LIN {X 0,Y 466.62,Z 631.984,A -85,B 0,C 180,E1 -7650.863,E2 -7650.863} C_VEL
LIN {X 0,Y 466.694,Z 631.335,A -85,B 0,C 180,E1 -7651.726,E2 -7651.726} C_VEL
LIN {X 0,Y 466.71,Z 630.282,A -85,B 0,C 180,E1 -7652.589,E2 -7652.589} C_VEL
LIN {X 0,Y 466.73,Z 628.811,A -85,B 0,C 180,E1 -7653.453,E2 -7653.453} C_VEL
LIN {X 0,Y 466.701,Z 625.736,A -85,B 0,C 180,E1 -7654.751,E2 -7654.751} C_VEL
LIN {X 0,Y 466.773,Z 621.588,A -85,B 0,C 180,E1 -7656.05,E2 -7656.05} C_VEL
LIN {X 0,Y 466.928,Z 615.211,A -85,B 0,C 180,E1 -7657.568,E2 -7657.568} C_VEL
LIN {X 0,Y 467.142,Z 608.264,A -85,B 0,C 180,E1 -7658.871,E2 -7658.871} C_VEL
LIN {X 0,Y 467.463,Z 599.648,A -85,B 0,C 180,E1 -7660.175,E2 -7660.175} C_VEL
LIN {X 0,Y 467.909,Z 590.815,A -85,B 0,C 180,E1 -7661.26,E2 -7661.26} C_VEL
LIN {X 0,Y 468.338,Z 580.643,A -85,B 0,C 180,E1 -7662.287,E2 -7662.287} C_VEL
LIN {X 0,Y 468.829,Z 569.32,A -85,B 0,C 180,E1 -7663.215,E2 -7663.215} C_VEL
LIN {X 0,Y 469.286,Z 557.554,A -85,B 0,C 180,E1 -7663.975,E2 -7663.975} C_VEL
LIN {X 0,Y 469.739,Z 544.43,A -85,B 0,C 180,E1 -7664.624,E2 -7664.624} C_VEL
LIN {X 0,Y 468.125,Z 531.649,A -85,B 0,C 180,E1 -7665.143,E2 -7665.143} C_VEL
LIN {X 0,Y 467.02,Z 523.223,A -85,B 0,C 180,E1 -7665.409,E2 -7665.409} C_VEL
LIN {X 0,Y 467.168,Z 513.678,A -85,B 0,C 180,E1 -7668.601,E2 -7668.601} C_VEL
LIN {X 0,Y 467.391,Z 504.9,A -85,B 0,C 180,E1 -7671.617,E2 -7671.617} C_VEL
LIN {X 0,Y 467.664,Z 495.775,A -85,B 0,C 180,E1 -7674.884,E2 -7674.884} C_VEL
LIN {X 0,Y 468.021,Z 488.237,A -85,B 0,C 180,E1 -7677.743,E2 -7677.743} C_VEL
LIN {X 0,Y 468.559,Z 479.713,A -85,B 0,C 180,E1 -7681.245,E2 -7681.245} C_VEL
LIN {X 0,Y 469.039,Z 474.432,A -85,B 0,C 180,E1 -7683.67,E2 -7683.67} C_VEL
LIN {X 0,Y 469.375,Z 469.859,A -85,B 0,C 180,E1 -7686.046,E2 -7686.046} C_VEL
LIN {X 0,Y 469.096,Z 466.887,A -85,B 0,C 180,E1 -7687.899,E2 -7687.899} C_VEL
LIN {X 0,Y 468.575,Z 463.943,A -85,B 0,C 180,E1 -7690.162,E2 -7690.162} C_VEL
LIN {X 0,Y 468.164,Z 461.563,A -85,B 0,C 180,E1 -7692.644,E2 -7692.644} C_VEL
LIN {X 0,Y 467.906,Z 460.071,A -85,B 0,C 180,E1 -7695.094,E2 -7695.094} C_VEL
LIN {X 0,Y 467.787,Z 459.398,A -85,B 0,C 180,E1 -7697.462,E2 -7697.462} C_VEL
LIN {X 0,Y 467.762,Z 459.412,A -85,B 0,C 180,E1 -7700.02,E2 -7700.02} C_VEL
LIN {X 0,Y 467.837,Z 460.213,A -85,B 0,C 180,E1 -7703.066,E2 -7703.066} C_VEL
LIN {X 0,Y 467.816,Z 461.445,A -85,B 0,C 180,E1 -7705.717,E2 -7705.717} C_VEL
LIN {X 0,Y 467.647,Z 462.959,A -85,B 0,C 180,E1 -7708.265,E2 -7708.265} C_VEL
LIN {X 0,Y 467.464,Z 465.049,A -85,B 0,C 180,E1 -7711.243,E2 -7711.243} C_VEL
LIN {X 0,Y 467.288,Z 467.552,A -85,B 0,C 180,E1 -7714.476,E2 -7714.476} C_VEL
LIN {X 0,Y 467.169,Z 469.646,A -85,B 0,C 180,E1 -7716.975,E2 -7716.975} C_VEL
LIN {X 0,Y 467.058,Z 472.089,A -85,B 0,C 180,E1 -7719.752,E2 -7719.752} C_VEL
LIN {X 0,Y 466.99,Z 474.598,A -85,B 0,C 180,E1 -7722.483,E2 -7722.483} C_VEL
LIN {X 0,Y 467.017,Z 476.743,A -85,B 0,C 180,E1 -7724.739,E2 -7724.739} C_VEL
LIN {X 0,Y 469.978,Z 489.42,A -85,B 0,C 180,E1 -7725.273,E2 -7725.273} C_VEL
LIN {X 0,Y 470.134,Z 495.785,A -85,B 0,C 180,E1 -7725.555,E2 -7725.555} C_VEL
LIN {X 0,Y 469.76,Z 507.117,A -85,B 0,C 180,E1 -7726.151,E2 -7726.151} C_VEL
LIN {X 0,Y 469.317,Z 518.894,A -85,B 0,C 180,E1 -7726.955,E2 -7726.955} C_VEL
LIN {X 0,Y 468.819,Z 529.714,A -85,B 0,C 180,E1 -7727.885,E2 -7727.885} C_VEL
LIN {X 0,Y 468.295,Z 539.912,A -85,B 0,C 180,E1 -7728.969,E2 -7728.969} C_VEL
LIN {X 0,Y 467.847,Z 549.675,A -85,B 0,C 180,E1 -7730.271,E2 -7730.271} C_VEL
LIN {X 0,Y 467.45,Z 557.526,A -85,B 0,C 180,E1 -7731.571,E2 -7731.571} C_VEL
LIN {X 0,Y 467.22,Z 562.822,A -85,B 0,C 180,E1 -7732.654,E2 -7732.654} C_VEL
LIN {X 0,Y 467.057,Z 567.987,A -85,B 0,C 180,E1 -7733.954,E2 -7733.954} C_VEL
LIN {X 0,Y 466.887,Z 571.984,A -85,B 0,C 180,E1 -7735.251,E2 -7735.251} C_VEL
LIN {X 0,Y 466.794,Z 574.921,A -85,B 0,C 180,E1 -7736.548,E2 -7736.548} C_VEL
LIN {X 0,Y 466.81,Z 576.332,A -85,B 0,C 180,E1 -7737.411,E2 -7737.411} C_VEL
LIN {X 0,Y 466.62,Z 577.923,A -85,B 0,C 180,E1 -7739.137,E2 -7739.137} C_VEL
LIN {X 0,Y 466.6,Z 578.133,A -85,B 0,C 180,E1 -7740,E2 -7740} C_VEL
LIN {X 0,Y 466.62,Z 577.913,A -85,B 0,C 180,E1 -7740.863,E2 -7740.863} C_VEL
LIN {X 0,Y 466.79,Z 576.267,A -85,B 0,C 180,E1 -7742.589,E2 -7742.589} C_VEL
LIN {X 0,Y 466.786,Z 574.855,A -85,B 0,C 180,E1 -7743.453,E2 -7743.453} C_VEL
LIN {X 0,Y 466.861,Z 571.894,A -85,B 0,C 180,E1 -7744.75,E2 -7744.75} C_VEL
LIN {X 0,Y 467.046,Z 567.886,A -85,B 0,C 180,E1 -7746.047,E2 -7746.047} C_VEL
LIN {X 0,Y 467.174,Z 562.727,A -85,B 0,C 180,E1 -7747.347,E2 -7747.347} C_VEL
LIN {X 0,Y 467.431,Z 556.22,A -85,B 0,C 180,E1 -7748.648,E2 -7748.648} C_VEL
LIN {X 0,Y 467.789,Z 548.123,A -85,B 0,C 180,E1 -7749.949,E2 -7749.949} C_VEL
LIN {X 0,Y 468.17,Z 539.866,A -85,B 0,C 180,E1 -7751.035,E2 -7751.035} C_VEL
LIN {X 0,Y 468.738,Z 529.781,A -85,B 0,C 180,E1 -7752.117,E2 -7752.117} C_VEL
LIN {X 0,Y 469.143,Z 518.266,A -85,B 0,C 180,E1 -7753.107,E2 -7753.107} C_VEL
LIN {X 0,Y 469.555,Z 507.32,A -85,B 0,C 180,E1 -7753.856,E2 -7753.856} C_VEL
LIN {X 0,Y 469.986,Z 495.028,A -85,B 0,C 180,E1 -7754.506,E2 -7754.506} C_VEL
LIN {X 0,Y 469.852,Z 489.361,A -85,B 0,C 180,E1 -7754.754,E2 -7754.754} C_VEL
LIN {X 0,Y 467.68,Z 478.772,A -85,B 0,C 180,E1 -7755.187,E2 -7755.187} C_VEL
LIN {X 0,Y 466.852,Z 474.833,A -85,B 0,C 180,E1 -7755.323,E2 -7755.323} C_VEL
LIN {X 0,Y 466.83,Z 471.352,A -85,B 0,C 180,E1 -7758.476,E2 -7758.476} C_VEL
LIN {X 0,Y 466.807,Z 468.406,A -85,B 0,C 180,E1 -7761.182,E2 -7761.182} C_VEL
LIN {X 0,Y 466.863,Z 465.394,A -85,B 0,C 180,E1 -7763.982,E2 -7763.982} C_VEL
LIN {X 0,Y 466.949,Z 462.367,A -85,B 0,C 180,E1 -7766.842,E2 -7766.842} C_VEL
LIN {X 0,Y 466.958,Z 459.297,A -85,B 0,C 180,E1 -7769.78,E2 -7769.78} C_VEL
LIN {X 0,Y 467.012,Z 458.315,A -85,B 0,C 180,E1 -7770.931,E2 -7770.931} C_VEL
LIN {X 0,Y 467.392,Z 458.268,A -85,B 0,C 180,E1 -7774.206,E2 -7774.206} C_VEL
LIN {X 0,Y 467.544,Z 458.245,A -85,B 0,C 180,E1 -7777.185,E2 -7777.185} C_VEL
LIN {X 0,Y 467.582,Z 458.242,A -85,B 0,C 180,E1 -7780.265,E2 -7780.265} C_VEL
LIN {X 0,Y 467.591,Z 458.241,A -85,B 0,C 180,E1 -7782.567,E2 -7782.567} C_VEL
LIN {X 0,Y 467.571,Z 458.241,A -85,B 0,C 180,E1 -7785.053,E2 -7785.053} C_VEL
LIN {X 0,Y 467.594,Z 458.239,A -85,B 0,C 180,E1 -7787.44,E2 -7787.44} C_VEL
LIN {X 0,Y 467.587,Z 458.241,A -85,B 0,C 180,E1 -7790.855,E2 -7790.855} C_VEL
LIN {X 0,Y 467.565,Z 458.245,A -85,B 0,C 180,E1 -7794.261,E2 -7794.261} C_VEL
LIN {X 0,Y 467.587,Z 458.241,A -85,B 0,C 180,E1 -7797.321,E2 -7797.321} C_VEL
LIN {X 0,Y 467.573,Z 458.241,A -85,B 0,C 180,E1 -7800.668,E2 -7800.668} C_VEL
LIN {X 0,Y 467.622,Z 458.237,A -85,B 0,C 180,E1 -7803.2,E2 -7803.2} C_VEL
LIN {X 0,Y 467.598,Z 458.241,A -85,B 0,C 180,E1 -7806.468,E2 -7806.468} C_VEL
LIN {X 0,Y 467.629,Z 458.238,A -85,B 0,C 180,E1 -7809.777,E2 -7809.777} C_VEL
LIN {X 0,Y 467.628,Z 458.236,A -85,B 0,C 180,E1 -7811.423,E2 -7811.423} C_VEL
LIN {X 0,Y 466.988,Z 458.317,A -85,B 0,C 180,E1 -7812.142,E2 -7812.142} C_VEL
LIN {X 0,Y 464.137,Z 458.669,A -85,B 0,C 180,E1 -7813.31,E2 -7813.31} C_VEL
LIN {X 0,Y 461.703,Z 458.976,A -85,B 0,C 180,E1 -7814.251,E2 -7814.251} C_VEL
LIN {X 0,Y 460.647,Z 459.103,A -85,B 0,C 180,E1 -7814.979,E2 -7814.979} C_VEL
LIN {X 0,Y 460.557,Z 459.114,A -85,B 0,C 180,E1 -7815.226,E2 -7815.226} C_VEL
LIN {X 0,Y 460.616,Z 459.111,A -85,B 0,C 180,E1 -7818.559,E2 -7818.559} C_VEL
LIN {X 0,Y 460.671,Z 459.105,A -85,B 0,C 180,E1 -7822.108,E2 -7822.108} C_VEL
LIN {X 0,Y 460.702,Z 459.099,A -85,B 0,C 180,E1 -7824.748,E2 -7824.748} C_VEL
LIN {X 0,Y 460.805,Z 459.085,A -85,B 0,C 180,E1 -7827.377,E2 -7827.377} C_VEL
LIN {X 0,Y 460.859,Z 459.081,A -85,B 0,C 180,E1 -7830,E2 -7830} C_VEL
LIN {X 0,Y 460.805,Z 459.087,A -85,B 0,C 180,E1 -7832.622,E2 -7832.622} C_VEL
LIN {X 0,Y 460.69,Z 459.102,A -85,B 0,C 180,E1 -7836.13,E2 -7836.13} C_VEL
LIN {X 0,Y 460.634,Z 459.107,A -85,B 0,C 180,E1 -7838.776,E2 -7838.776} C_VEL
LIN {X 0,Y 460.619,Z 459.109,A -85,B 0,C 180,E1 -7842.445,E2 -7842.445} C_VEL
LIN {X 0,Y 460.605,Z 459.111,A -85,B 0,C 180,E1 -7845.997,E2 -7845.997} C_VEL
LIN {X 0,Y 460.576,Z 459.114,A -85,B 0,C 180,E1 -7848.901,E2 -7848.901} C_VEL
LIN {X 0,Y 460.521,Z 459.121,A -85,B 0,C 180,E1 -7851.485,E2 -7851.485} C_VEL
LIN {X 0,Y 460.546,Z 459.119,A -85,B 0,C 180,E1 -7854.332,E2 -7854.332} C_VEL
LIN {X 0,Y 460.577,Z 459.112,A -85,B 0,C 180,E1 -7857.243,E2 -7857.243} C_VEL
LIN {X 0,Y 460.515,Z 459.121,A -85,B 0,C 180,E1 -7860.24,E2 -7860.24} C_VEL
LIN {X 0,Y 460.533,Z 459.119,A -85,B 0,C 180,E1 -7863.324,E2 -7863.324} C_VEL
LIN {X 0,Y 460.482,Z 459.124,A -85,B 0,C 180,E1 -7866.529,E2 -7866.529} C_VEL
LIN {X 0,Y 460.548,Z 459.118,A -85,B 0,C 180,E1 -7868.897,E2 -7868.897} C_VEL
LIN {X 0,Y 460.526,Z 459.12,A -85,B 0,C 180,E1 -7872.181,E2 -7872.181} C_VEL
LIN {X 0,Y 460.523,Z 459.122,A -85,B 0,C 180,E1 -7875.412,E2 -7875.412} C_VEL
LIN {X 0,Y 460.538,Z 459.118,A -85,B 0,C 180,E1 -7878.397,E2 -7878.397} C_VEL
LIN {X 0,Y 460.521,Z 459.122,A -85,B 0,C 180,E1 -7881.266,E2 -7881.266} C_VEL
LIN {X 0,Y 460.516,Z 459.121,A -85,B 0,C 180,E1 -7884.554,E2 -7884.554} C_VEL
LIN {X 0,Y 460.534,Z 459.121,A -85,B 0,C 180,E1 -7887.715,E2 -7887.715} C_VEL
LIN {X 0,Y 460.542,Z 459.119,A -85,B 0,C 180,E1 -7890.769,E2 -7890.769} C_VEL
LIN {X 0,Y 460.565,Z 459.118,A -85,B 0,C 180,E1 -7893.734,E2 -7893.734} C_VEL
LIN {X 0,Y 460.547,Z 459.118,A -85,B 0,C 180,E1 -7896.624,E2 -7896.624} C_VEL
LIN {X 0,Y 460.554,Z 459.117,A -85,B 0,C 180,E1 -7899.453,E2 -7899.453} C_VEL
LIN {X 0,Y 460.561,Z 459.114,A -85,B 0,C 180,E1 -7902.23,E2 -7902.23} C_VEL
LIN {X 0,Y 460.567,Z 459.117,A -85,B 0,C 180,E1 -7904.965,E2 -7904.965} C_VEL
LIN {X 0,Y 460.613,Z 459.106,A -85,B 0,C 180,E1 -7908.559,E2 -7908.559} C_VEL
LIN {X 0,Y 460.696,Z 459.101,A -85,B 0,C 180,E1 -7912.108,E2 -7912.108} C_VEL
LIN {X 0,Y 460.698,Z 459.097,A -85,B 0,C 180,E1 -7914.748,E2 -7914.748} C_VEL
LIN {X 0,Y 460.825,Z 459.085,A -85,B 0,C 180,E1 -7917.377,E2 -7917.377} C_VEL
LIN {X 0,Y 460.855,Z 459.081,A -85,B 0,C 180,E1 -7920,E2 -7920} C_VEL
LIN {X 0,Y 460.801,Z 459.084,A -85,B 0,C 180,E1 -7922.622,E2 -7922.622} C_VEL
LIN {X 0,Y 460.711,Z 459.098,A -85,B 0,C 180,E1 -7926.13,E2 -7926.13} C_VEL
LIN {X 0,Y 460.629,Z 459.106,A -85,B 0,C 180,E1 -7928.776,E2 -7928.776} C_VEL
LIN {X 0,Y 460.614,Z 459.109,A -85,B 0,C 180,E1 -7932.445,E2 -7932.445} C_VEL
LIN {X 0,Y 460.601,Z 459.111,A -85,B 0,C 180,E1 -7935.997,E2 -7935.997} C_VEL
LIN {X 0,Y 460.572,Z 459.115,A -85,B 0,C 180,E1 -7938.902,E2 -7938.902} C_VEL
LIN {X 0,Y 460.516,Z 459.122,A -85,B 0,C 180,E1 -7941.486,E2 -7941.486} C_VEL
LIN {X 0,Y 460.543,Z 459.115,A -85,B 0,C 180,E1 -7944.332,E2 -7944.332} C_VEL
LIN {X 0,Y 460.58,Z 459.114,A -85,B 0,C 180,E1 -7947.243,E2 -7947.243} C_VEL
LIN {X 0,Y 460.511,Z 459.121,A -85,B 0,C 180,E1 -7950.24,E2 -7950.24} C_VEL
LIN {X 0,Y 460.529,Z 459.121,A -85,B 0,C 180,E1 -7953.325,E2 -7953.325} C_VEL
LIN {X 0,Y 460.479,Z 459.127,A -85,B 0,C 180,E1 -7956.529,E2 -7956.529} C_VEL
LIN {X 0,Y 460.545,Z 459.117,A -85,B 0,C 180,E1 -7958.898,E2 -7958.898} C_VEL
LIN {X 0,Y 460.547,Z 459.118,A -85,B 0,C 180,E1 -7962.179,E2 -7962.179} C_VEL
LIN {X 0,Y 460.514,Z 459.128,A -85,B 0,C 180,E1 -7965.411,E2 -7965.411} C_VEL
LIN {X 0,Y 460.532,Z 459.124,A -85,B 0,C 180,E1 -7968.398,E2 -7968.398} C_VEL
LIN {X 0,Y 460.565,Z 459.206,A -85,B 0,C 180,E1 -7969.188,E2 -7969.188} C_VEL
LIN {X 0,Y 461.793,Z 466.092,A -85,B 0,C 180,E1 -7972.315,E2 -7972.315} C_VEL
LIN {X 0,Y 462.377,Z 470.478,A -85,B 0,C 180,E1 -7974.209,E2 -7974.209} C_VEL
LIN {X 0,Y 462.014,Z 476.847,A -85,B 0,C 180,E1 -7976.796,E2 -7976.796} C_VEL
LIN {X 0,Y 461.551,Z 484.581,A -85,B 0,C 180,E1 -7979.835,E2 -7979.835} C_VEL
LIN {X 0,Y 461.107,Z 492.34,A -85,B 0,C 180,E1 -7982.791,E2 -7982.791} C_VEL
LIN {X 0,Y 460.773,Z 500.11,A -85,B 0,C 180,E1 -7985.681,E2 -7985.681} C_VEL
LIN {X 0,Y 460.386,Z 509.336,A -85,B 0,C 180,E1 -7989.025,E2 -7989.025} C_VEL
LIN {X 0,Y 460.159,Z 517.005,A -85,B 0,C 180,E1 -7991.754,E2 -7991.754} C_VEL
LIN {X 0,Y 460.033,Z 524.604,A -85,B 0,C 180,E1 -7994.406,E2 -7994.406} C_VEL
LIN {X 0,Y 461.907,Z 538.263,A -85,B 0,C 180,E1 -7994.853,E2 -7994.853} C_VEL
LIN {X 0,Y 462.917,Z 546.399,A -85,B 0,C 180,E1 -7995.212,E2 -7995.212} C_VEL
LIN {X 0,Y 462.482,Z 558.305,A -85,B 0,C 180,E1 -7995.816,E2 -7995.816} C_VEL
LIN {X 0,Y 461.956,Z 569.987,A -85,B 0,C 180,E1 -7996.585,E2 -7996.585} C_VEL
LIN {X 0,Y 461.407,Z 581.292,A -85,B 0,C 180,E1 -7997.534,E2 -7997.534} C_VEL
LIN {X 0,Y 460.931,Z 591.248,A -85,B 0,C 180,E1 -7998.567,E2 -7998.567} C_VEL
LIN {X 0,Y 460.462,Z 599.965,A -85,B 0,C 180,E1 -7999.669,E2 -7999.669} C_VEL
LIN {X 0,Y 460.108,Z 608.449,A -85,B 0,C 180,E1 -8000.993,E2 -8000.993} C_VEL
LIN {X 0,Y 459.867,Z 615.276,A -85,B 0,C 180,E1 -8002.315,E2 -8002.315} C_VEL
LIN {X 0,Y 459.677,Z 621.541,A -85,B 0,C 180,E1 -8003.856,E2 -8003.856} C_VEL
LIN {X 0,Y 459.631,Z 625.603,A -85,B 0,C 180,E1 -8005.176,E2 -8005.176} C_VEL
LIN {X 0,Y 459.627,Z 628.592,A -85,B 0,C 180,E1 -8006.494,E2 -8006.494} C_VEL
LIN {X 0,Y 459.621,Z 630.019,A -85,B 0,C 180,E1 -8007.371,E2 -8007.371} C_VEL
LIN {X 0,Y 459.629,Z 631.023,A -85,B 0,C 180,E1 -8008.248,E2 -8008.248} C_VEL
LIN {X 0,Y 459.553,Z 631.62,A -85,B 0,C 180,E1 -8009.124,E2 -8009.124} C_VEL
LIN {X 0,Y 459.529,Z 631.819,A -85,B 0,C 180,E1 -8010,E2 -8010} C_VEL
LIN {X 0,Y 459.553,Z 631.571,A -85,B 0,C 180,E1 -8010.876,E2 -8010.876} C_VEL
LIN {X 0,Y 459.631,Z 630.919,A -85,B 0,C 180,E1 -8011.753,E2 -8011.753} C_VEL
LIN {X 0,Y 459.63,Z 629.858,A -85,B 0,C 180,E1 -8012.629,E2 -8012.629} C_VEL
LIN {X 0,Y 459.643,Z 628.379,A -85,B 0,C 180,E1 -8013.507,E2 -8013.507} C_VEL
LIN {X 0,Y 459.632,Z 625.289,A -85,B 0,C 180,E1 -8014.824,E2 -8014.824} C_VEL
LIN {X 0,Y 459.714,Z 620.037,A -85,B 0,C 180,E1 -8016.431,E2 -8016.431} C_VEL
LIN {X 0,Y 459.895,Z 613.684,A -85,B 0,C 180,E1 -8017.905,E2 -8017.905} C_VEL
LIN {X 0,Y 460.181,Z 606.485,A -85,B 0,C 180,E1 -8019.228,E2 -8019.228} C_VEL
LIN {X 0,Y 460.507,Z 597.482,A -85,B 0,C 180,E1 -8020.553,E2 -8020.553} C_VEL
LIN {X 0,Y 461.071,Z 587.326,A -85,B 0,C 180,E1 -8021.764,E2 -8021.764} C_VEL
LIN {X 0,Y 461.488,Z 576.916,A -85,B 0,C 180,E1 -8022.767,E2 -8022.767} C_VEL
LIN {X 0,Y 462.034,Z 565.747,A -85,B 0,C 180,E1 -8023.637,E2 -8023.637} C_VEL
LIN {X 0,Y 462.589,Z 553.269,A -85,B 0,C 180,E1 -8024.406,E2 -8024.406} C_VEL
LIN {X 0,Y 462.819,Z 545.368,A -85,B 0,C 180,E1 -8024.792,E2 -8024.792} C_VEL
LIN {X 0,Y 461.169,Z 531.714,A -85,B 0,C 180,E1 -8025.377,E2 -8025.377} C_VEL
LIN {X 0,Y 459.944,Z 522.74,A -85,B 0,C 180,E1 -8025.664,E2 -8025.664} C_VEL
LIN {X 0,Y 460.125,Z 512.626,A -85,B 0,C 180,E1 -8029.125,E2 -8029.125} C_VEL
LIN {X 0,Y 460.346,Z 504.578,A -85,B 0,C 180,E1 -8031.965,E2 -8031.965} C_VEL
LIN {X 0,Y 460.679,Z 495.558,A -85,B 0,C 180,E1 -8035.288,E2 -8035.288} C_VEL
LIN {X 0,Y 461.042,Z 488.122,A -85,B 0,C 180,E1 -8038.201,E2 -8038.201} C_VEL
LIN {X 0,Y 461.592,Z 480.372,A -85,B 0,C 180,E1 -8041.501,E2 -8041.501} C_VEL
LIN {X 0,Y 462.144,Z 474.635,A -85,B 0,C 180,E1 -8044.241,E2 -8044.241} C_VEL
LIN {X 0,Y 462.399,Z 470.78,A -85,B 0,C 180,E1 -8046.353,E2 -8046.353} C_VEL
LIN {X 0,Y 462.013,Z 467.441,A -85,B 0,C 180,E1 -8048.586,E2 -8048.586} C_VEL
LIN {X 0,Y 461.529,Z 464.7,A -85,B 0,C 180,E1 -8050.904,E2 -8050.904} C_VEL
LIN {X 0,Y 461.142,Z 462.652,A -85,B 0,C 180,E1 -8053.3,E2 -8053.3} C_VEL
LIN {X 0,Y 460.922,Z 461.348,A -85,B 0,C 180,E1 -8055.778,E2 -8055.778} C_VEL
LIN {X 0,Y 460.826,Z 460.803,A -85,B 0,C 180,E1 -8058.357,E2 -8058.357} C_VEL
LIN {X 0,Y 460.804,Z 461.042,A -85,B 0,C 180,E1 -8061.295,E2 -8061.295} C_VEL
LIN {X 0,Y 460.87,Z 461.851,A -85,B 0,C 180,E1 -8063.923,E2 -8063.923} C_VEL
LIN {X 0,Y 460.746,Z 463.376,A -85,B 0,C 180,E1 -8067.029,E2 -8067.029} C_VEL
LIN {X 0,Y 460.511,Z 465.551,A -85,B 0,C 180,E1 -8070.447,E2 -8070.447} C_VEL
LIN {X 0,Y 460.288,Z 467.945,A -85,B 0,C 180,E1 -8073.718,E2 -8073.718} C_VEL
LIN {X 0,Y 460.182,Z 470.267,A -85,B 0,C 180,E1 -8076.604,E2 -8076.604} C_VEL
LIN {X 0,Y 460.019,Z 472.686,A -85,B 0,C 180,E1 -8079.428,E2 -8079.428} C_VEL
LIN {X 0,Y 459.946,Z 475.184,A -85,B 0,C 180,E1 -8082.206,E2 -8082.206} C_VEL
LIN {X 0,Y 459.946,Z 477.301,A -85,B 0,C 180,E1 -8084.471,E2 -8084.471} C_VEL
LIN {X 0,Y 463.097,Z 490.22,A -85,B 0,C 180,E1 -8085.049,E2 -8085.049} C_VEL
LIN {X 0,Y 463.31,Z 495.315,A -85,B 0,C 180,E1 -8085.281,E2 -8085.281} C_VEL
LIN {X 0,Y 462.917,Z 507.758,A -85,B 0,C 180,E1 -8085.942,E2 -8085.942} C_VEL
LIN {X 0,Y 462.437,Z 518.485,A -85,B 0,C 180,E1 -8086.677,E2 -8086.677} C_VEL
LIN {X 0,Y 461.906,Z 530.268,A -85,B 0,C 180,E1 -8087.701,E2 -8087.701} C_VEL
LIN {X 0,Y 461.344,Z 540.431,A -85,B 0,C 180,E1 -8088.8,E2 -8088.8} C_VEL
LIN {X 0,Y 460.868,Z 550.145,A -85,B 0,C 180,E1 -8090.122,E2 -8090.122} C_VEL
LIN {X 0,Y 460.438,Z 557.967,A -85,B 0,C 180,E1 -8091.442,E2 -8091.442} C_VEL
LIN {X 0,Y 460.186,Z 563.247,A -85,B 0,C 180,E1 -8092.541,E2 -8092.541} C_VEL
LIN {X 0,Y 460.016,Z 568.417,A -85,B 0,C 180,E1 -8093.861,E2 -8093.861} C_VEL
LIN {X 0,Y 459.83,Z 572.417,A -85,B 0,C 180,E1 -8095.178,E2 -8095.178} C_VEL
LIN {X 0,Y 459.733,Z 575.353,A -85,B 0,C 180,E1 -8096.494,E2 -8096.494} C_VEL
LIN {X 0,Y 459.736,Z 576.763,A -85,B 0,C 180,E1 -8097.372,E2 -8097.372} C_VEL
LIN {X 0,Y 459.554,Z 578.344,A -85,B 0,C 180,E1 -8099.124,E2 -8099.124} C_VEL
LIN {X 0,Y 459.531,Z 578.549,A -85,B 0,C 180,E1 -8100,E2 -8100} C_VEL
LIN {X 0,Y 459.554,Z 578.319,A -85,B 0,C 180,E1 -8100.876,E2 -8100.876} C_VEL
LIN {X 0,Y 459.637,Z 577.682,A -85,B 0,C 180,E1 -8101.753,E2 -8101.753} C_VEL
LIN {X 0,Y 459.705,Z 576.654,A -85,B 0,C 180,E1 -8102.629,E2 -8102.629} C_VEL
LIN {X 0,Y 459.726,Z 575.229,A -85,B 0,C 180,E1 -8103.506,E2 -8103.506} C_VEL
LIN {X 0,Y 459.79,Z 572.247,A -85,B 0,C 180,E1 -8104.823,E2 -8104.823} C_VEL
LIN {X 0,Y 460.005,Z 568.213,A -85,B 0,C 180,E1 -8106.14,E2 -8106.14} C_VEL
LIN {X 0,Y 460.157,Z 562.011,A -85,B 0,C 180,E1 -8107.68,E2 -8107.68} C_VEL
LIN {X 0,Y 460.504,Z 555.24,A -85,B 0,C 180,E1 -8109,E2 -8109} C_VEL
LIN {X 0,Y 460.886,Z 546.841,A -85,B 0,C 180,E1 -8110.322,E2 -8110.322} C_VEL
LIN {X 0,Y 461.275,Z 538.195,A -85,B 0,C 180,E1 -8111.424,E2 -8111.424} C_VEL
LIN {X 0,Y 461.901,Z 527.691,A -85,B 0,C 180,E1 -8112.512,E2 -8112.512} C_VEL
LIN {X 0,Y 462.279,Z 517.091,A -85,B 0,C 180,E1 -8113.406,E2 -8113.406} C_VEL
LIN {X 0,Y 462.749,Z 505.515,A -85,B 0,C 180,E1 -8114.176,E2 -8114.176} C_VEL
LIN {X 0,Y 463.204,Z 492.473,A -85,B 0,C 180,E1 -8114.835,E2 -8114.835} C_VEL
LIN {X 0,Y 461.989,Z 485.133,A -85,B 0,C 180,E1 -8115.169,E2 -8115.169} C_VEL
LIN {X 0,Y 459.762,Z 475.138,A -85,B 0,C 180,E1 -8115.574,E2 -8115.574} C_VEL
LIN {X 0,Y 459.736,Z 471.673,A -85,B 0,C 180,E1 -8118.725,E2 -8118.725} C_VEL
LIN {X 0,Y 459.744,Z 468.648,A -85,B 0,C 180,E1 -8121.524,E2 -8121.524} C_VEL
LIN {X 0,Y 459.805,Z 465.601,A -85,B 0,C 180,E1 -8124.374,E2 -8124.374} C_VEL
LIN {X 0,Y 459.917,Z 462.535,A -85,B 0,C 180,E1 -8127.286,E2 -8127.286} C_VEL
LIN {X 0,Y 459.904,Z 459.428,A -85,B 0,C 180,E1 -8130.285,E2 -8130.285} C_VEL
LIN {X 0,Y 460.173,Z 459.167,A -85,B 0,C 180,E1 -8132.861,E2 -8132.861} C_VEL
LIN {X 0,Y 460.439,Z 459.132,A -85,B 0,C 180,E1 -8135.452,E2 -8135.452} C_VEL
LIN {X 0,Y 460.548,Z 459.116,A -85,B 0,C 180,E1 -8138.898,E2 -8138.898} C_VEL
LIN {X 0,Y 460.528,Z 459.12,A -85,B 0,C 180,E1 -8142.181,E2 -8142.181} C_VEL
LIN {X 0,Y 460.519,Z 459.119,A -85,B 0,C 180,E1 -8145.411,E2 -8145.411} C_VEL
LIN {X 0,Y 460.537,Z 459.119,A -85,B 0,C 180,E1 -8148.398,E2 -8148.398} C_VEL
LIN {X 0,Y 460.532,Z 459.119,A -85,B 0,C 180,E1 -8151.267,E2 -8151.267} C_VEL
LIN {X 0,Y 460.516,Z 459.121,A -85,B 0,C 180,E1 -8154.554,E2 -8154.554} C_VEL
LIN {X 0,Y 460.537,Z 459.119,A -85,B 0,C 180,E1 -8157.716,E2 -8157.716} C_VEL
LIN {X 0,Y 460.543,Z 459.116,A -85,B 0,C 180,E1 -8160.769,E2 -8160.769} C_VEL
LIN {X 0,Y 460.569,Z 459.116,A -85,B 0,C 180,E1 -8163.735,E2 -8163.735} C_VEL
LIN {X 0,Y 460.552,Z 459.117,A -85,B 0,C 180,E1 -8166.624,E2 -8166.624} C_VEL
LIN {X 0,Y 460.557,Z 459.117,A -85,B 0,C 180,E1 -8169.453,E2 -8169.453} C_VEL
LIN {X 0,Y 460.563,Z 459.117,A -85,B 0,C 180,E1 -8172.23,E2 -8172.23} C_VEL
LIN {X 0,Y 460.572,Z 459.112,A -85,B 0,C 180,E1 -8174.965,E2 -8174.965} C_VEL
LIN {X 0,Y 460.557,Z 459.114,A -85,B 0,C 180,E1 -8175.226,E2 -8175.226} C_VEL
LIN {X 0,Y 459.879,Z 459.203,A -85,B 0,C 180,E1 -8175.956,E2 -8175.956} C_VEL
LIN {X 0,Y 457.031,Z 459.555,A -85,B 0,C 180,E1 -8177.142,E2 -8177.142} C_VEL
LIN {X 0,Y 454.634,Z 459.854,A -85,B 0,C 180,E1 -8178.099,E2 -8178.099} C_VEL
LIN {X 0,Y 453.612,Z 459.982,A -85,B 0,C 180,E1 -8178.838,E2 -8178.838} C_VEL
LIN {X 0,Y 453.532,Z 459.991,A -85,B 0,C 180,E1 -8179.088,E2 -8179.088} C_VEL
LIN {X 0,Y 453.66,Z 459.974,A -85,B 0,C 180,E1 -8182.517,E2 -8182.517} C_VEL
LIN {X 0,Y 453.676,Z 459.974,A -85,B 0,C 180,E1 -8184.667,E2 -8184.667} C_VEL
LIN {X 0,Y 453.749,Z 459.964,A -85,B 0,C 180,E1 -8187.337,E2 -8187.337} C_VEL
LIN {X 0,Y 453.829,Z 459.957,A -85,B 0,C 180,E1 -8190,E2 -8190} C_VEL
LIN {X 0,Y 453.749,Z 459.965,A -85,B 0,C 180,E1 -8192.663,E2 -8192.663} C_VEL
LIN {X 0,Y 453.656,Z 459.977,A -85,B 0,C 180,E1 -8196.225,E2 -8196.225} C_VEL
LIN {X 0,Y 453.598,Z 459.983,A -85,B 0,C 180,E1 -8198.913,E2 -8198.913} C_VEL
LIN {X 0,Y 453.569,Z 459.986,A -85,B 0,C 180,E1 -8202.529,E2 -8202.529} C_VEL
LIN {X 0,Y 453.55,Z 459.989,A -85,B 0,C 180,E1 -8206.196,E2 -8206.196} C_VEL
LIN {X 0,Y 453.525,Z 459.992,A -85,B 0,C 180,E1 -8209.04,E2 -8209.04} C_VEL
LIN {X 0,Y 453.481,Z 460,A -85,B 0,C 180,E1 -8211.836,E2 -8211.836} C_VEL
LIN {X 0,Y 453.518,Z 459.993,A -85,B 0,C 180,E1 -8214.734,E2 -8214.734} C_VEL
LIN {X 0,Y 453.536,Z 459.993,A -85,B 0,C 180,E1 -8217.959,E2 -8217.959} C_VEL
LIN {X 0,Y 453.47,Z 460,A -85,B 0,C 180,E1 -8221.525,E2 -8221.525} C_VEL
LIN {X 0,Y 453.493,Z 459.994,A -85,B 0,C 180,E1 -8224.777,E2 -8224.777} C_VEL
LIN {X 0,Y 453.476,Z 459.999,A -85,B 0,C 180,E1 -8228.31,E2 -8228.31} C_VEL
LIN {X 0,Y 453.497,Z 459.995,A -85,B 0,C 180,E1 -8230.608,E2 -8230.608} C_VEL
LIN {X 0,Y 453.459,Z 460,A -85,B 0,C 180,E1 -8233.244,E2 -8233.244} C_VEL
LIN {X 0,Y 453.476,Z 459.999,A -85,B 0,C 180,E1 -8235.78,E2 -8235.78} C_VEL
LIN {X 0,Y 453.484,Z 459.998,A -85,B 0,C 180,E1 -8238.209,E2 -8238.209} C_VEL
LIN {X 0,Y 453.49,Z 459.995,A -85,B 0,C 180,E1 -8240.794,E2 -8240.794} C_VEL
LIN {X 0,Y 453.459,Z 460.001,A -85,B 0,C 180,E1 -8243.917,E2 -8243.917} C_VEL
LIN {X 0,Y 453.485,Z 459.996,A -85,B 0,C 180,E1 -8247.151,E2 -8247.151} C_VEL
LIN {X 0,Y 453.477,Z 460,A -85,B 0,C 180,E1 -8250.268,E2 -8250.268} C_VEL
LIN {X 0,Y 453.511,Z 459.994,A -85,B 0,C 180,E1 -8253.294,E2 -8253.294} C_VEL
LIN {X 0,Y 453.504,Z 459.995,A -85,B 0,C 180,E1 -8256.238,E2 -8256.238} C_VEL
LIN {X 0,Y 453.484,Z 459.997,A -85,B 0,C 180,E1 -8259.117,E2 -8259.117} C_VEL
LIN {X 0,Y 453.514,Z 459.993,A -85,B 0,C 180,E1 -8261.944,E2 -8261.944} C_VEL
LIN {X 0,Y 453.541,Z 459.99,A -85,B 0,C 180,E1 -8264.726,E2 -8264.726} C_VEL
LIN {X 0,Y 453.561,Z 459.985,A -85,B 0,C 180,E1 -8268.379,E2 -8268.379} C_VEL
LIN {X 0,Y 453.653,Z 459.977,A -85,B 0,C 180,E1 -8271.985,E2 -8271.985} C_VEL
LIN {X 0,Y 453.672,Z 459.973,A -85,B 0,C 180,E1 -8274.667,E2 -8274.667} C_VEL
LIN {X 0,Y 453.765,Z 459.965,A -85,B 0,C 180,E1 -8277.337,E2 -8277.337} C_VEL
LIN {X 0,Y 453.825,Z 459.957,A -85,B 0,C 180,E1 -8280,E2 -8280} C_VEL
LIN {X 0,Y 453.745,Z 459.962,A -85,B 0,C 180,E1 -8282.663,E2 -8282.663} C_VEL
LIN {X 0,Y 453.678,Z 459.974,A -85,B 0,C 180,E1 -8286.225,E2 -8286.225} C_VEL
LIN {X 0,Y 453.593,Z 459.983,A -85,B 0,C 180,E1 -8288.913,E2 -8288.913} C_VEL
LIN {X 0,Y 453.564,Z 459.987,A -85,B 0,C 180,E1 -8292.529,E2 -8292.529} C_VEL
LIN {X 0,Y 453.545,Z 459.989,A -85,B 0,C 180,E1 -8296.196,E2 -8296.196} C_VEL
LIN {X 0,Y 453.522,Z 459.995,A -85,B 0,C 180,E1 -8299.041,E2 -8299.041} C_VEL
LIN {X 0,Y 453.477,Z 460,A -85,B 0,C 180,E1 -8301.836,E2 -8301.836} C_VEL
LIN {X 0,Y 453.515,Z 459.992,A -85,B 0,C 180,E1 -8304.734,E2 -8304.734} C_VEL
LIN {X 0,Y 453.538,Z 459.992,A -85,B 0,C 180,E1 -8307.961,E2 -8307.961} C_VEL
LIN {X 0,Y 453.466,Z 460.001,A -85,B 0,C 180,E1 -8311.525,E2 -8311.525} C_VEL
LIN {X 0,Y 453.489,Z 459.998,A -85,B 0,C 180,E1 -8314.778,E2 -8314.778} C_VEL
LIN {X 0,Y 453.473,Z 459.997,A -85,B 0,C 180,E1 -8318.311,E2 -8318.311} C_VEL
LIN {X 0,Y 453.495,Z 459.996,A -85,B 0,C 180,E1 -8320.609,E2 -8320.609} C_VEL
LIN {X 0,Y 453.481,Z 459.998,A -85,B 0,C 180,E1 -8323.248,E2 -8323.248} C_VEL
LIN {X 0,Y 453.464,Z 460.006,A -85,B 0,C 180,E1 -8325.779,E2 -8325.779} C_VEL
LIN {X 0,Y 453.523,Z 460.168,A -85,B 0,C 180,E1 -8328.969,E2 -8328.969} C_VEL
LIN {X 0,Y 454.718,Z 466.78,A -85,B 0,C 180,E1 -8332.022,E2 -8332.022} C_VEL
LIN {X 0,Y 455.375,Z 471.468,A -85,B 0,C 180,E1 -8334.093,E2 -8334.093} C_VEL
LIN {X 0,Y 455.063,Z 477.317,A -85,B 0,C 180,E1 -8336.51,E2 -8336.51} C_VEL
LIN {X 0,Y 454.474,Z 486.054,A -85,B 0,C 180,E1 -8339.996,E2 -8339.996} C_VEL
LIN {X 0,Y 454.07,Z 493.377,A -85,B 0,C 180,E1 -8342.833,E2 -8342.833} C_VEL
LIN {X 0,Y 453.627,Z 502.427,A -85,B 0,C 180,E1 -8346.246,E2 -8346.246} C_VEL
LIN {X 0,Y 453.247,Z 511.485,A -85,B 0,C 180,E1 -8349.581,E2 -8349.581} C_VEL
LIN {X 0,Y 453.035,Z 519.269,A -85,B 0,C 180,E1 -8352.392,E2 -8352.392} C_VEL
LIN {X 0,Y 452.937,Z 524.455,A -85,B 0,C 180,E1 -8354.177,E2 -8354.177} C_VEL
LIN {X 0,Y 454.88,Z 538.291,A -85,B 0,C 180,E1 -8354.645,E2 -8354.645} C_VEL
LIN {X 0,Y 455.973,Z 548.142,A -85,B 0,C 180,E1 -8355.096,E2 -8355.096} C_VEL
LIN {X 0,Y 455.47,Z 559.531,A -85,B 0,C 180,E1 -8355.707,E2 -8355.707} C_VEL
LIN {X 0,Y 454.925,Z 570.79,A -85,B 0,C 180,E1 -8356.487,E2 -8356.487} C_VEL
LIN {X 0,Y 454.346,Z 582.32,A -85,B 0,C 180,E1 -8357.493,E2 -8357.493} C_VEL
LIN {X 0,Y 453.815,Z 592.606,A -85,B 0,C 180,E1 -8358.612,E2 -8358.612} C_VEL
LIN {X 0,Y 453.291,Z 602.488,A -85,B 0,C 180,E1 -8359.955,E2 -8359.955} C_VEL
LIN {X 0,Y 452.976,Z 610.446,A -85,B 0,C 180,E1 -8361.299,E2 -8361.299} C_VEL
LIN {X 0,Y 452.757,Z 615.837,A -85,B 0,C 180,E1 -8362.418,E2 -8362.418} C_VEL
LIN {X 0,Y 452.603,Z 621.102,A -85,B 0,C 180,E1 -8363.76,E2 -8363.76} C_VEL
LIN {X 0,Y 452.561,Z 625.176,A -85,B 0,C 180,E1 -8365.1,E2 -8365.1} C_VEL
LIN {X 0,Y 452.527,Z 628.172,A -85,B 0,C 180,E1 -8366.439,E2 -8366.439} C_VEL
LIN {X 0,Y 452.543,Z 629.607,A -85,B 0,C 180,E1 -8367.33,E2 -8367.33} C_VEL
LIN {X 0,Y 452.538,Z 630.611,A -85,B 0,C 180,E1 -8368.22,E2 -8368.22} C_VEL
LIN {X 0,Y 452.489,Z 631.21,A -85,B 0,C 180,E1 -8369.11,E2 -8369.11} C_VEL
LIN {X 0,Y 452.463,Z 631.408,A -85,B 0,C 180,E1 -8370,E2 -8370} C_VEL
LIN {X 0,Y 452.489,Z 631.16,A -85,B 0,C 180,E1 -8370.89,E2 -8370.89} C_VEL
LIN {X 0,Y 452.539,Z 630.501,A -85,B 0,C 180,E1 -8371.78,E2 -8371.78} C_VEL
LIN {X 0,Y 452.552,Z 629.438,A -85,B 0,C 180,E1 -8372.671,E2 -8372.671} C_VEL
LIN {X 0,Y 452.541,Z 627.952,A -85,B 0,C 180,E1 -8373.562,E2 -8373.562} C_VEL
LIN {X 0,Y 452.562,Z 624.857,A -85,B 0,C 180,E1 -8374.9,E2 -8374.9} C_VEL
LIN {X 0,Y 452.628,Z 620.029,A -85,B 0,C 180,E1 -8376.416,E2 -8376.416} C_VEL
LIN {X 0,Y 452.841,Z 613.225,A -85,B 0,C 180,E1 -8378.029,E2 -8378.029} C_VEL
LIN {X 0,Y 453.113,Z 606.022,A -85,B 0,C 180,E1 -8379.373,E2 -8379.373} C_VEL
LIN {X 0,Y 453.495,Z 597.027,A -85,B 0,C 180,E1 -8380.718,E2 -8380.718} C_VEL
LIN {X 0,Y 454.025,Z 586.87,A -85,B 0,C 180,E1 -8381.949,E2 -8381.949} C_VEL
LIN {X 0,Y 454.498,Z 576.497,A -85,B 0,C 180,E1 -8382.967,E2 -8382.967} C_VEL
LIN {X 0,Y 455.161,Z 563.828,A -85,B 0,C 180,E1 -8383.961,E2 -8383.961} C_VEL
LIN {X 0,Y 455.773,Z 550.894,A -85,B 0,C 180,E1 -8384.74,E2 -8384.74} C_VEL
LIN {X 0,Y 455.768,Z 545.225,A -85,B 0,C 180,E1 -8385.026,E2 -8385.026} C_VEL
LIN {X 0,Y 454.238,Z 531.252,A -85,B 0,C 180,E1 -8385.642,E2 -8385.642} C_VEL
LIN {X 0,Y 452.873,Z 522.188,A -85,B 0,C 180,E1 -8385.964,E2 -8385.964} C_VEL
LIN {X 0,Y 453.088,Z 512.14,A -85,B 0,C 180,E1 -8389.481,E2 -8389.481} C_VEL
LIN {X 0,Y 453.313,Z 504.286,A -85,B 0,C 180,E1 -8392.324,E2 -8392.324} C_VEL
LIN {X 0,Y 453.687,Z 495.371,A -85,B 0,C 180,E1 -8395.706,E2 -8395.706} C_VEL
LIN {X 0,Y 454.089,Z 488.049,A -85,B 0,C 180,E1 -8398.672,E2 -8398.672} C_VEL
LIN {X 0,Y 454.644,Z 481.025,A -85,B 0,C 180,E1 -8401.766,E2 -8401.766} C_VEL
LIN {X 0,Y 455.19,Z 475.881,A -85,B 0,C 180,E1 -8404.302,E2 -8404.302} C_VEL
LIN {X 0,Y 455.421,Z 471.776,A -85,B 0,C 180,E1 -8406.634,E2 -8406.634} C_VEL
LIN {X 0,Y 455.186,Z 469.546,A -85,B 0,C 180,E1 -8408.141,E2 -8408.141} C_VEL
LIN {X 0,Y 454.636,Z 466.415,A -85,B 0,C 180,E1 -8410.758,E2 -8410.758} C_VEL
LIN {X 0,Y 454.228,Z 464.193,A -85,B 0,C 180,E1 -8413.347,E2 -8413.347} C_VEL
LIN {X 0,Y 453.998,Z 462.868,A -85,B 0,C 180,E1 -8415.844,E2 -8415.844} C_VEL
LIN {X 0,Y 453.884,Z 462.305,A -85,B 0,C 180,E1 -8418.255,E2 -8418.255} C_VEL
LIN {X 0,Y 453.832,Z 462.349,A -85,B 0,C 180,E1 -8420.742,E2 -8420.742} C_VEL
LIN {X 0,Y 453.901,Z 463.163,A -85,B 0,C 180,E1 -8423.958,E2 -8423.958} C_VEL
LIN {X 0,Y 453.729,Z 464.652,A -85,B 0,C 180,E1 -8427.171,E2 -8427.171} C_VEL
LIN {X 0,Y 453.517,Z 466.534,A -85,B 0,C 180,E1 -8430.271,E2 -8430.271} C_VEL
LIN {X 0,Y 453.268,Z 468.652,A -85,B 0,C 180,E1 -8433.279,E2 -8433.279} C_VEL
LIN {X 0,Y 453.131,Z 470.925,A -85,B 0,C 180,E1 -8436.218,E2 -8436.218} C_VEL
LIN {X 0,Y 453.021,Z 473.31,A -85,B 0,C 180,E1 -8439.095,E2 -8439.095} C_VEL
LIN {X 0,Y 452.917,Z 475.787,A -85,B 0,C 180,E1 -8441.92,E2 -8441.92} C_VEL
LIN {X 0,Y 452.935,Z 477.86,A -85,B 0,C 180,E1 -8444.192,E2 -8444.192} C_VEL
LIN {X 0,Y 455.998,Z 490.097,A -85,B 0,C 180,E1 -8444.754,E2 -8444.754} C_VEL
LIN {X 0,Y 456.601,Z 493.935,A -85,B 0,C 180,E1 -8444.946,E2 -8444.946} C_VEL
LIN {X 0,Y 456.131,Z 506.666,A -85,B 0,C 180,E1 -8445.614,E2 -8445.614} C_VEL
LIN {X 0,Y 455.636,Z 517.509,A -85,B 0,C 180,E1 -8446.35,E2 -8446.35} C_VEL
LIN {X 0,Y 455.138,Z 528.529,A -85,B 0,C 180,E1 -8447.289,E2 -8447.289} C_VEL
LIN {X 0,Y 454.455,Z 539.081,A -85,B 0,C 180,E1 -8448.402,E2 -8448.402} C_VEL
LIN {X 0,Y 454.071,Z 547.677,A -85,B 0,C 180,E1 -8449.522,E2 -8449.522} C_VEL
LIN {X 0,Y 453.632,Z 556.048,A -85,B 0,C 180,E1 -8450.863,E2 -8450.863} C_VEL
LIN {X 0,Y 453.294,Z 561.762,A -85,B 0,C 180,E1 -8451.979,E2 -8451.979} C_VEL
LIN {X 0,Y 453.033,Z 567.784,A -85,B 0,C 180,E1 -8453.454,E2 -8453.454} C_VEL
LIN {X 0,Y 452.776,Z 572.874,A -85,B 0,C 180,E1 -8455.103,E2 -8455.103} C_VEL
LIN {X 0,Y 452.676,Z 575.795,A -85,B 0,C 180,E1 -8456.44,E2 -8456.44} C_VEL
LIN {X 0,Y 452.652,Z 577.197,A -85,B 0,C 180,E1 -8457.33,E2 -8457.33} C_VEL
LIN {X 0,Y 452.579,Z 578.174,A -85,B 0,C 180,E1 -8458.22,E2 -8458.22} C_VEL
LIN {X 0,Y 452.465,Z 578.964,A -85,B 0,C 180,E1 -8460,E2 -8460} C_VEL
LIN {X 0,Y 452.49,Z 578.725,A -85,B 0,C 180,E1 -8460.89,E2 -8460.89} C_VEL
LIN {X 0,Y 452.577,Z 578.077,A -85,B 0,C 180,E1 -8461.78,E2 -8461.78} C_VEL
LIN {X 0,Y 452.624,Z 577.04,A -85,B 0,C 180,E1 -8462.67,E2 -8462.67} C_VEL
LIN {X 0,Y 452.667,Z 575.601,A -85,B 0,C 180,E1 -8463.561,E2 -8463.561} C_VEL
LIN {X 0,Y 452.704,Z 572.6,A -85,B 0,C 180,E1 -8464.898,E2 -8464.898} C_VEL
LIN {X 0,Y 453.014,Z 567.487,A -85,B 0,C 180,E1 -8466.525,E2 -8466.525} C_VEL
LIN {X 0,Y 453.181,Z 561.277,A -85,B 0,C 180,E1 -8468.023,E2 -8468.023} C_VEL
LIN {X 0,Y 453.554,Z 554.236,A -85,B 0,C 180,E1 -8469.364,E2 -8469.364} C_VEL
LIN {X 0,Y 454.018,Z 545.421,A -85,B 0,C 180,E1 -8470.705,E2 -8470.705} C_VEL
LIN {X 0,Y 454.503,Z 535.436,A -85,B 0,C 180,E1 -8471.936,E2 -8471.936} C_VEL
LIN {X 0,Y 455.034,Z 525.889,A -85,B 0,C 180,E1 -8472.887,E2 -8472.887} C_VEL
LIN {X 0,Y 455.485,Z 514.709,A -85,B 0,C 180,E1 -8473.792,E2 -8473.792} C_VEL
LIN {X 0,Y 455.959,Z 503.597,A -85,B 0,C 180,E1 -8474.506,E2 -8474.506} C_VEL
LIN {X 0,Y 456.273,Z 492.431,A -85,B 0,C 180,E1 -8475.066,E2 -8475.066} C_VEL
LIN {X 0,Y 453.614,Z 479.529,A -85,B 0,C 180,E1 -8475.635,E2 -8475.635} C_VEL
LIN {X 0,Y 452.655,Z 475.465,A -85,B 0,C 180,E1 -8475.81,E2 -8475.81} C_VEL
LIN {X 0,Y 452.645,Z 471.949,A -85,B 0,C 180,E1 -8479.03,E2 -8479.03} C_VEL
LIN {X 0,Y 452.672,Z 468.879,A -85,B 0,C 180,E1 -8481.877,E2 -8481.877} C_VEL
LIN {X 0,Y 452.744,Z 465.801,A -85,B 0,C 180,E1 -8484.78,E2 -8484.78} C_VEL
LIN {X 0,Y 452.816,Z 462.656,A -85,B 0,C 180,E1 -8487.788,E2 -8487.788} C_VEL
LIN {X 0,Y 452.824,Z 460.617,A -85,B 0,C 180,E1 -8489.779,E2 -8489.779} C_VEL
LIN {X 0,Y 452.971,Z 460.063,A -85,B 0,C 180,E1 -8491.422,E2 -8491.422} C_VEL
LIN {X 0,Y 453.356,Z 460.015,A -85,B 0,C 180,E1 -8494.753,E2 -8494.753} C_VEL
LIN {X 0,Y 453.451,Z 460,A -85,B 0,C 180,E1 -8497.772,E2 -8497.772} C_VEL
LIN {X 0,Y 453.499,Z 459.995,A -85,B 0,C 180,E1 -8500.609,E2 -8500.609} C_VEL
LIN {X 0,Y 453.46,Z 460,A -85,B 0,C 180,E1 -8503.244,E2 -8503.244} C_VEL
LIN {X 0,Y 453.468,Z 459.998,A -85,B 0,C 180,E1 -8505.779,E2 -8505.779} C_VEL
LIN {X 0,Y 453.484,Z 459.998,A -85,B 0,C 180,E1 -8508.209,E2 -8508.209} C_VEL
LIN {X 0,Y 453.515,Z 459.994,A -85,B 0,C 180,E1 -8510.791,E2 -8510.791} C_VEL
LIN {X 0,Y 453.46,Z 460.002,A -85,B 0,C 180,E1 -8513.917,E2 -8513.917} C_VEL
LIN {X 0,Y 453.488,Z 459.997,A -85,B 0,C 180,E1 -8517.151,E2 -8517.151} C_VEL
LIN {X 0,Y 453.479,Z 460,A -85,B 0,C 180,E1 -8520.268,E2 -8520.268} C_VEL
LIN {X 0,Y 453.512,Z 459.994,A -85,B 0,C 180,E1 -8523.294,E2 -8523.294} C_VEL
LIN {X 0,Y 453.509,Z 459.997,A -85,B 0,C 180,E1 -8526.239,E2 -8526.239} C_VEL
LIN {X 0,Y 453.488,Z 459.996,A -85,B 0,C 180,E1 -8529.118,E2 -8529.118} C_VEL
LIN {X 0,Y 453.516,Z 459.993,A -85,B 0,C 180,E1 -8531.945,E2 -8531.945} C_VEL
LIN {X 0,Y 453.546,Z 459.988,A -85,B 0,C 180,E1 -8534.726,E2 -8534.726} C_VEL
LIN {X 0,Y 453.565,Z 459.988,A -85,B 0,C 180,E1 -8538.379,E2 -8538.379} C_VEL
LIN {X 0,Y 453.532,Z 459.991,A -85,B 0,C 180,E1 -8539.088,E2 -8539.088} C_VEL
LIN {X 0,Y 452.878,Z 460.074,A -85,B 0,C 180,E1 -8539.829,E2 -8539.829} C_VEL
LIN {X 0,Y 450.052,Z 460.426,A -85,B 0,C 180,E1 -8541.034,E2 -8541.034} C_VEL
LIN {X 0,Y 447.669,Z 460.725,A -85,B 0,C 180,E1 -8542.006,E2 -8542.006} C_VEL
LIN {X 0,Y 446.664,Z 460.845,A -85,B 0,C 180,E1 -8542.757,E2 -8542.757} C_VEL
LIN {X 0,Y 446.592,Z 460.854,A -85,B 0,C 180,E1 -8543.011,E2 -8543.011} C_VEL
LIN {X 0,Y 446.65,Z 460.849,A -85,B 0,C 180,E1 -8544.582,E2 -8544.582} C_VEL
LIN {X 0,Y 446.67,Z 460.849,A -85,B 0,C 180,E1 -8548.196,E2 -8548.196} C_VEL
LIN {X 0,Y 446.799,Z 460.832,A -85,B 0,C 180,E1 -8550,E2 -8550} C_VEL
LIN {X 0,Y 446.696,Z 460.843,A -85,B 0,C 180,E1 -8552.705,E2 -8552.705} C_VEL
LIN {X 0,Y 446.624,Z 460.852,A -85,B 0,C 180,E1 -8556.324,E2 -8556.324} C_VEL
LIN {X 0,Y 446.544,Z 460.862,A -85,B 0,C 180,E1 -8559.055,E2 -8559.055} C_VEL
LIN {X 0,Y 446.527,Z 460.862,A -85,B 0,C 180,E1 -8562.729,E2 -8562.729} C_VEL
LIN {X 0,Y 446.501,Z 460.867,A -85,B 0,C 180,E1 -8566.228,E2 -8566.228} C_VEL
LIN {X 0,Y 446.474,Z 460.87,A -85,B 0,C 180,E1 -8569.303,E2 -8569.303} C_VEL
LIN {X 0,Y 446.423,Z 460.877,A -85,B 0,C 180,E1 -8572.199,E2 -8572.199} C_VEL
LIN {X 0,Y 446.462,Z 460.873,A -85,B 0,C 180,E1 -8575.152,E2 -8575.152} C_VEL
LIN {X 0,Y 446.489,Z 460.869,A -85,B 0,C 180,E1 -8578.178,E2 -8578.178} C_VEL
LIN {X 0,Y 446.423,Z 460.877,A -85,B 0,C 180,E1 -8581.775,E2 -8581.775} C_VEL
LIN {X 0,Y 446.434,Z 460.874,A -85,B 0,C 180,E1 -8584.522,E2 -8584.522} C_VEL
LIN {X 0,Y 446.434,Z 460.876,A -85,B 0,C 180,E1 -8588.081,E2 -8588.081} C_VEL
LIN {X 0,Y 446.43,Z 460.875,A -85,B 0,C 180,E1 -8590.917,E2 -8590.917} C_VEL
LIN {X 0,Y 446.405,Z 460.88,A -85,B 0,C 180,E1 -8593.845,E2 -8593.845} C_VEL
LIN {X 0,Y 446.424,Z 460.878,A -85,B 0,C 180,E1 -8596.4,E2 -8596.4} C_VEL
LIN {X 0,Y 446.444,Z 460.877,A -85,B 0,C 180,E1 -8599.802,E2 -8599.802} C_VEL
LIN {X 0,Y 446.411,Z 460.88,A -85,B 0,C 180,E1 -8603.255,E2 -8603.255} C_VEL
LIN {X 0,Y 446.45,Z 460.871,A -85,B 0,C 180,E1 -8606.566,E2 -8606.566} C_VEL
LIN {X 0,Y 446.433,Z 460.876,A -85,B 0,C 180,E1 -8609.979,E2 -8609.979} C_VEL
LIN {X 0,Y 446.481,Z 460.869,A -85,B 0,C 180,E1 -8612.839,E2 -8612.839} C_VEL
LIN {X 0,Y 446.466,Z 460.871,A -85,B 0,C 180,E1 -8615.923,E2 -8615.923} C_VEL
LIN {X 0,Y 446.455,Z 460.873,A -85,B 0,C 180,E1 -8618.773,E2 -8618.773} C_VEL
LIN {X 0,Y 446.46,Z 460.875,A -85,B 0,C 180,E1 -8621.649,E2 -8621.649} C_VEL
LIN {X 0,Y 446.509,Z 460.866,A -85,B 0,C 180,E1 -8624.479,E2 -8624.479} C_VEL
LIN {X 0,Y 446.519,Z 460.863,A -85,B 0,C 180,E1 -8628.193,E2 -8628.193} C_VEL
LIN {X 0,Y 446.602,Z 460.855,A -85,B 0,C 180,E1 -8631.858,E2 -8631.858} C_VEL
LIN {X 0,Y 446.646,Z 460.848,A -85,B 0,C 180,E1 -8634.582,E2 -8634.582} C_VEL
LIN {X 0,Y 446.709,Z 460.844,A -85,B 0,C 180,E1 -8637.294,E2 -8637.294} C_VEL
LIN {X 0,Y 446.795,Z 460.832,A -85,B 0,C 180,E1 -8640,E2 -8640} C_VEL
LIN {X 0,Y 446.692,Z 460.841,A -85,B 0,C 180,E1 -8642.705,E2 -8642.705} C_VEL
LIN {X 0,Y 446.648,Z 460.849,A -85,B 0,C 180,E1 -8646.323,E2 -8646.323} C_VEL
LIN {X 0,Y 446.538,Z 460.862,A -85,B 0,C 180,E1 -8649.055,E2 -8649.055} C_VEL
LIN {X 0,Y 446.522,Z 460.865,A -85,B 0,C 180,E1 -8652.73,E2 -8652.73} C_VEL
LIN {X 0,Y 446.497,Z 460.866,A -85,B 0,C 180,E1 -8656.228,E2 -8656.228} C_VEL
LIN {X 0,Y 446.47,Z 460.873,A -85,B 0,C 180,E1 -8659.303,E2 -8659.303} C_VEL
LIN {X 0,Y 446.419,Z 460.877,A -85,B 0,C 180,E1 -8662.199,E2 -8662.199} C_VEL
LIN {X 0,Y 446.459,Z 460.874,A -85,B 0,C 180,E1 -8665.152,E2 -8665.152} C_VEL
LIN {X 0,Y 446.485,Z 460.869,A -85,B 0,C 180,E1 -8668.179,E2 -8668.179} C_VEL
LIN {X 0,Y 446.419,Z 460.877,A -85,B 0,C 180,E1 -8671.775,E2 -8671.775} C_VEL
LIN {X 0,Y 446.431,Z 460.876,A -85,B 0,C 180,E1 -8674.523,E2 -8674.523} C_VEL
LIN {X 0,Y 446.431,Z 460.874,A -85,B 0,C 180,E1 -8678.082,E2 -8678.082} C_VEL
LIN {X 0,Y 446.432,Z 460.878,A -85,B 0,C 180,E1 -8680.918,E2 -8680.918} C_VEL
LIN {X 0,Y 446.444,Z 460.877,A -85,B 0,C 180,E1 -8683.841,E2 -8683.841} C_VEL
LIN {X 0,Y 446.399,Z 460.885,A -85,B 0,C 180,E1 -8686.404,E2 -8686.404} C_VEL
LIN {X 0,Y 446.483,Z 460.991,A -85,B 0,C 180,E1 -8688.68,E2 -8688.68} C_VEL
LIN {X 0,Y 447.622,Z 467.449,A -85,B 0,C 180,E1 -8691.724,E2 -8691.724} C_VEL
LIN {X 0,Y 448.368,Z 472.516,A -85,B 0,C 180,E1 -8693.999,E2 -8693.999} C_VEL
LIN {X 0,Y 447.992,Z 478.937,A -85,B 0,C 180,E1 -8696.697,E2 -8696.697} C_VEL
LIN {X 0,Y 447.468,Z 486.657,A -85,B 0,C 180,E1 -8699.828,E2 -8699.828} C_VEL
LIN {X 0,Y 447.018,Z 494.376,A -85,B 0,C 180,E1 -8702.875,E2 -8702.875} C_VEL
LIN {X 0,Y 446.622,Z 502.198,A -85,B 0,C 180,E1 -8705.879,E2 -8705.879} C_VEL
LIN {X 0,Y 446.204,Z 511.16,A -85,B 0,C 180,E1 -8709.244,E2 -8709.244} C_VEL
LIN {X 0,Y 445.967,Z 518.918,A -85,B 0,C 180,E1 -8712.104,E2 -8712.104} C_VEL
LIN {X 0,Y 445.878,Z 523.905,A -85,B 0,C 180,E1 -8713.925,E2 -8713.925} C_VEL
LIN {X 0,Y 447.934,Z 538.637,A -85,B 0,C 180,E1 -8714.45,E2 -8714.45} C_VEL
LIN {X 0,Y 449.032,Z 548.533,A -85,B 0,C 180,E1 -8714.918,E2 -8714.918} C_VEL
LIN {X 0,Y 448.449,Z 560.545,A -85,B 0,C 180,E1 -8715.594,E2 -8715.594} C_VEL
LIN {X 0,Y 447.863,Z 572.688,A -85,B 0,C 180,E1 -8716.482,E2 -8716.482} C_VEL
LIN {X 0,Y 447.226,Z 583.94,A -85,B 0,C 180,E1 -8717.521,E2 -8717.521} C_VEL
LIN {X 0,Y 446.706,Z 593.813,A -85,B 0,C 180,E1 -8718.658,E2 -8718.658} C_VEL
LIN {X 0,Y 446.171,Z 603.414,A -85,B 0,C 180,E1 -8720.022,E2 -8720.022} C_VEL
LIN {X 0,Y 445.873,Z 611.07,A -85,B 0,C 180,E1 -8721.388,E2 -8721.388} C_VEL
LIN {X 0,Y 445.615,Z 617.224,A -85,B 0,C 180,E1 -8722.752,E2 -8722.752} C_VEL
LIN {X 0,Y 445.494,Z 621.499,A -85,B 0,C 180,E1 -8723.927,E2 -8723.927} C_VEL
LIN {X 0,Y 445.43,Z 625.818,A -85,B 0,C 180,E1 -8725.475,E2 -8725.475} C_VEL
LIN {X 0,Y 445.428,Z 627.732,A -85,B 0,C 180,E1 -8726.382,E2 -8726.382} C_VEL
LIN {X 0,Y 445.467,Z 629.182,A -85,B 0,C 180,E1 -8727.287,E2 -8727.287} C_VEL
LIN {X 0,Y 445.45,Z 630.189,A -85,B 0,C 180,E1 -8728.192,E2 -8728.192} C_VEL
LIN {X 0,Y 445.426,Z 630.793,A -85,B 0,C 180,E1 -8729.096,E2 -8729.096} C_VEL
LIN {X 0,Y 445.399,Z 630.994,A -85,B 0,C 180,E1 -8730,E2 -8730} C_VEL
LIN {X 0,Y 445.427,Z 630.75,A -85,B 0,C 180,E1 -8730.904,E2 -8730.904} C_VEL
LIN {X 0,Y 445.452,Z 630.087,A -85,B 0,C 180,E1 -8731.808,E2 -8731.808} C_VEL
LIN {X 0,Y 445.475,Z 629.021,A -85,B 0,C 180,E1 -8732.713,E2 -8732.713} C_VEL
LIN {X 0,Y 445.441,Z 627.534,A -85,B 0,C 180,E1 -8733.619,E2 -8733.619} C_VEL
LIN {X 0,Y 445.492,Z 624.435,A -85,B 0,C 180,E1 -8734.978,E2 -8734.978} C_VEL
LIN {X 0,Y 445.529,Z 620.095,A -85,B 0,C 180,E1 -8736.386,E2 -8736.386} C_VEL
LIN {X 0,Y 445.72,Z 613.844,A -85,B 0,C 180,E1 -8737.93,E2 -8737.93} C_VEL
LIN {X 0,Y 446.023,Z 606.881,A -85,B 0,C 180,E1 -8739.295,E2 -8739.295} C_VEL
LIN {X 0,Y 446.378,Z 598.276,A -85,B 0,C 180,E1 -8740.661,E2 -8740.661} C_VEL
LIN {X 0,Y 446.945,Z 589.465,A -85,B 0,C 180,E1 -8741.796,E2 -8741.796} C_VEL
LIN {X 0,Y 447.33,Z 581.057,A -85,B 0,C 180,E1 -8742.707,E2 -8742.707} C_VEL
LIN {X 0,Y 447.965,Z 569.588,A -85,B 0,C 180,E1 -8743.727,E2 -8743.727} C_VEL
LIN {X 0,Y 448.518,Z 558.523,A -85,B 0,C 180,E1 -8744.52,E2 -8744.52} C_VEL
LIN {X 0,Y 448.916,Z 546.474,A -85,B 0,C 180,E1 -8745.203,E2 -8745.203} C_VEL
LIN {X 0,Y 447.344,Z 531.72,A -85,B 0,C 180,E1 -8745.89,E2 -8745.89} C_VEL
LIN {X 0,Y 445.803,Z 521.638,A -85,B 0,C 180,E1 -8746.273,E2 -8746.273} C_VEL
LIN {X 0,Y 446.04,Z 511.803,A -85,B 0,C 180,E1 -8749.802,E2 -8749.802} C_VEL
LIN {X 0,Y 446.277,Z 504.022,A -85,B 0,C 180,E1 -8752.695,E2 -8752.695} C_VEL
LIN {X 0,Y 446.711,Z 494.896,A -85,B 0,C 180,E1 -8756.263,E2 -8756.263} C_VEL
LIN {X 0,Y 447.141,Z 488.006,A -85,B 0,C 180,E1 -8759.16,E2 -8759.16} C_VEL
LIN {X 0,Y 447.734,Z 481.259,A -85,B 0,C 180,E1 -8762.256,E2 -8762.256} C_VEL
LIN {X 0,Y 448.245,Z 477.12,A -85,B 0,C 180,E1 -8764.364,E2 -8764.364} C_VEL
LIN {X 0,Y 448.436,Z 472.773,A -85,B 0,C 180,E1 -8766.938,E2 -8766.938} C_VEL
LIN {X 0,Y 448.084,Z 470.124,A -85,B 0,C 180,E1 -8768.858,E2 -8768.858} C_VEL
LIN {X 0,Y 447.608,Z 467.475,A -85,B 0,C 180,E1 -8771.258,E2 -8771.258} C_VEL
LIN {X 0,Y 447.236,Z 465.498,A -85,B 0,C 180,E1 -8773.744,E2 -8773.744} C_VEL
LIN {X 0,Y 447.039,Z 464.239,A -85,B 0,C 180,E1 -8776.318,E2 -8776.318} C_VEL
LIN {X 0,Y 446.918,Z 463.727,A -85,B 0,C 180,E1 -8779.01,E2 -8779.01} C_VEL
LIN {X 0,Y 446.915,Z 463.993,A -85,B 0,C 180,E1 -8782.172,E2 -8782.172} C_VEL
LIN {X 0,Y 446.878,Z 464.806,A -85,B 0,C 180,E1 -8784.865,E2 -8784.865} C_VEL
LIN {X 0,Y 446.676,Z 466.128,A -85,B 0,C 180,E1 -8787.659,E2 -8787.659} C_VEL
LIN {X 0,Y 446.44,Z 468.005,A -85,B 0,C 180,E1 -8790.79,E2 -8790.79} C_VEL
LIN {X 0,Y 446.227,Z 470.124,A -85,B 0,C 180,E1 -8793.863,E2 -8793.863} C_VEL
LIN {X 0,Y 446.051,Z 472.375,A -85,B 0,C 180,E1 -8796.803,E2 -8796.803} C_VEL
LIN {X 0,Y 445.922,Z 474.764,A -85,B 0,C 180,E1 -8799.712,E2 -8799.712} C_VEL
LIN {X 0,Y 445.848,Z 477.249,A -85,B 0,C 180,E1 -8802.572,E2 -8802.572} C_VEL
LIN {X 0,Y 445.882,Z 478.544,A -85,B 0,C 180,E1 -8803.894,E2 -8803.894} C_VEL
LIN {X 0,Y 449.063,Z 490.483,A -85,B 0,C 180,E1 -8804.475,E2 -8804.475} C_VEL
LIN {X 0,Y 449.824,Z 495.06,A -85,B 0,C 180,E1 -8804.713,E2 -8804.713} C_VEL
LIN {X 0,Y 449.321,Z 507.604,A -85,B 0,C 180,E1 -8805.391,E2 -8805.391} C_VEL
LIN {X 0,Y 448.804,Z 518.378,A -85,B 0,C 180,E1 -8806.141,E2 -8806.141} C_VEL
LIN {X 0,Y 448.25,Z 529.269,A -85,B 0,C 180,E1 -8807.092,E2 -8807.092} C_VEL
LIN {X 0,Y 447.53,Z 539.704,A -85,B 0,C 180,E1 -8808.22,E2 -8808.22} C_VEL
LIN {X 0,Y 447.115,Z 548.229,A -85,B 0,C 180,E1 -8809.357,E2 -8809.357} C_VEL
LIN {X 0,Y 446.651,Z 556.56,A -85,B 0,C 180,E1 -8810.719,E2 -8810.719} C_VEL
LIN {X 0,Y 446.268,Z 562.268,A -85,B 0,C 180,E1 -8811.852,E2 -8811.852} C_VEL
LIN {X 0,Y 445.998,Z 567.404,A -85,B 0,C 180,E1 -8813.099,E2 -8813.099} C_VEL
LIN {X 0,Y 445.662,Z 572.148,A -85,B 0,C 180,E1 -8814.571,E2 -8814.571} C_VEL
LIN {X 0,Y 445.765,Z 574.413,A -85,B 0,C 180,E1 -8815.479,E2 -8815.479} C_VEL
LIN {X 0,Y 445.621,Z 576.267,A -85,B 0,C 180,E1 -8816.383,E2 -8816.383} C_VEL
LIN {X 0,Y 445.572,Z 577.656,A -85,B 0,C 180,E1 -8817.288,E2 -8817.288} C_VEL
LIN {X 0,Y 445.521,Z 578.623,A -85,B 0,C 180,E1 -8818.192,E2 -8818.192} C_VEL
LIN {X 0,Y 445.401,Z 579.386,A -85,B 0,C 180,E1 -8820,E2 -8820} C_VEL
LIN {X 0,Y 445.428,Z 579.128,A -85,B 0,C 180,E1 -8820.904,E2 -8820.904} C_VEL
LIN {X 0,Y 445.502,Z 578.469,A -85,B 0,C 180,E1 -8821.808,E2 -8821.808} C_VEL
LIN {X 0,Y 445.546,Z 577.421,A -85,B 0,C 180,E1 -8822.713,E2 -8822.713} C_VEL
LIN {X 0,Y 445.608,Z 575.96,A -85,B 0,C 180,E1 -8823.617,E2 -8823.617} C_VEL
LIN {X 0,Y 445.622,Z 572.935,A -85,B 0,C 180,E1 -8824.976,E2 -8824.976} C_VEL
LIN {X 0,Y 445.91,Z 568.843,A -85,B 0,C 180,E1 -8826.334,E2 -8826.334} C_VEL
LIN {X 0,Y 446.089,Z 562.56,A -85,B 0,C 180,E1 -8827.924,E2 -8827.924} C_VEL
LIN {X 0,Y 446.471,Z 555.719,A -85,B 0,C 180,E1 -8829.285,E2 -8829.285} C_VEL
LIN {X 0,Y 446.939,Z 547.213,A -85,B 0,C 180,E1 -8830.648,E2 -8830.648} C_VEL
LIN {X 0,Y 447.354,Z 538.472,A -85,B 0,C 180,E1 -8831.785,E2 -8831.785} C_VEL
LIN {X 0,Y 447.981,Z 528.198,A -85,B 0,C 180,E1 -8832.875,E2 -8832.875} C_VEL
LIN {X 0,Y 448.415,Z 517.696,A -85,B 0,C 180,E1 -8833.785,E2 -8833.785} C_VEL
LIN {X 0,Y 448.986,Z 505.388,A -85,B 0,C 180,E1 -8834.62,E2 -8834.62} C_VEL
LIN {X 0,Y 449.361,Z 493.421,A -85,B 0,C 180,E1 -8835.245,E2 -8835.245} C_VEL
LIN {X 0,Y 446.618,Z 480.352,A -85,B 0,C 180,E1 -8835.84,E2 -8835.84} C_VEL
LIN {X 0,Y 445.56,Z 475.833,A -85,B 0,C 180,E1 -8836.015,E2 -8836.015} C_VEL
LIN {X 0,Y 445.574,Z 472.212,A -85,B 0,C 180,E1 -8839.344,E2 -8839.344} C_VEL
LIN {X 0,Y 445.584,Z 469.11,A -85,B 0,C 180,E1 -8842.244,E2 -8842.244} C_VEL
LIN {X 0,Y 445.681,Z 465.996,A -85,B 0,C 180,E1 -8845.2,E2 -8845.2} C_VEL
LIN {X 0,Y 445.758,Z 462.864,A -85,B 0,C 180,E1 -8848.229,E2 -8848.229} C_VEL
LIN {X 0,Y 445.774,Z 460.961,A -85,B 0,C 180,E1 -8850.299,E2 -8850.299} C_VEL
LIN {X 0,Y 446.153,Z 460.911,A -85,B 0,C 180,E1 -8853.459,E2 -8853.459} C_VEL
LIN {X 0,Y 446.346,Z 460.887,A -85,B 0,C 180,E1 -8855.633,E2 -8855.633} C_VEL
LIN {X 0,Y 446.448,Z 460.872,A -85,B 0,C 180,E1 -8859.027,E2 -8859.027} C_VEL
LIN {X 0,Y 446.439,Z 460.875,A -85,B 0,C 180,E1 -8862.277,E2 -8862.277} C_VEL
LIN {X 0,Y 446.456,Z 460.871,A -85,B 0,C 180,E1 -8865.104,E2 -8865.104} C_VEL
LIN {X 0,Y 446.433,Z 460.876,A -85,B 0,C 180,E1 -8868.609,E2 -8868.609} C_VEL
LIN {X 0,Y 446.462,Z 460.872,A -85,B 0,C 180,E1 -8870.974,E2 -8870.974} C_VEL
LIN {X 0,Y 446.424,Z 460.877,A -85,B 0,C 180,E1 -8874.374,E2 -8874.374} C_VEL
LIN {X 0,Y 446.427,Z 460.877,A -85,B 0,C 180,E1 -8877.639,E2 -8877.639} C_VEL
LIN {X 0,Y 446.453,Z 460.872,A -85,B 0,C 180,E1 -8880.791,E2 -8880.791} C_VEL
LIN {X 0,Y 446.483,Z 460.87,A -85,B 0,C 180,E1 -8883.848,E2 -8883.848} C_VEL
LIN {X 0,Y 446.435,Z 460.874,A -85,B 0,C 180,E1 -8886.823,E2 -8886.823} C_VEL
LIN {X 0,Y 446.45,Z 460.876,A -85,B 0,C 180,E1 -8889.737,E2 -8889.737} C_VEL
LIN {X 0,Y 446.468,Z 460.872,A -85,B 0,C 180,E1 -8892.597,E2 -8892.597} C_VEL
LIN {X 0,Y 446.477,Z 460.869,A -85,B 0,C 180,E1 -8895.412,E2 -8895.412} C_VEL
LIN {X 0,Y 446.523,Z 460.865,A -85,B 0,C 180,E1 -8898.193,E2 -8898.193} C_VEL
LIN {X 0,Y 446.538,Z 460.861,A -85,B 0,C 180,E1 -8900.944,E2 -8900.944} C_VEL
LIN {X 0,Y 446.592,Z 460.854,A -85,B 0,C 180,E1 -8903.011,E2 -8903.011} C_VEL
LIN {X 0,Y 445.92,Z 460.942,A -85,B 0,C 180,E1 -8903.763,E2 -8903.763} C_VEL
LIN {X 0,Y 442.975,Z 461.306,A -85,B 0,C 180,E1 -8904.984,E2 -8904.984} C_VEL
LIN {X 0,Y 440.543,Z 461.61,A -85,B 0,C 180,E1 -8905.969,E2 -8905.969} C_VEL
LIN {X 0,Y 439.597,Z 461.727,A -85,B 0,C 180,E1 -8906.731,E2 -8906.731} C_VEL
LIN {X 0,Y 439.573,Z 461.729,A -85,B 0,C 180,E1 -8906.989,E2 -8906.989} C_VEL
LIN {X 0,Y 439.768,Z 461.708,A -85,B 0,C 180,E1 -8910,E2 -8910} C_VEL
LIN {X 0,Y 439.645,Z 461.721,A -85,B 0,C 180,E1 -8912.749,E2 -8912.749} C_VEL
LIN {X 0,Y 439.596,Z 461.726,A -85,B 0,C 180,E1 -8916.425,E2 -8916.425} C_VEL
LIN {X 0,Y 439.506,Z 461.739,A -85,B 0,C 180,E1 -8919.201,E2 -8919.201} C_VEL
LIN {X 0,Y 439.471,Z 461.741,A -85,B 0,C 180,E1 -8922.937,E2 -8922.937} C_VEL
LIN {X 0,Y 439.452,Z 461.746,A -85,B 0,C 180,E1 -8926.348,E2 -8926.348} C_VEL
LIN {X 0,Y 439.407,Z 461.751,A -85,B 0,C 180,E1 -8929.626,E2 -8929.626} C_VEL
LIN {X 0,Y 439.37,Z 461.755,A -85,B 0,C 180,E1 -8932.575,E2 -8932.575} C_VEL
LIN {X 0,Y 439.409,Z 461.751,A -85,B 0,C 180,E1 -8935.584,E2 -8935.584} C_VEL
LIN {X 0,Y 439.421,Z 461.747,A -85,B 0,C 180,E1 -8938.673,E2 -8938.673} C_VEL
LIN {X 0,Y 439.374,Z 461.756,A -85,B 0,C 180,E1 -8942.03,E2 -8942.03} C_VEL
LIN {X 0,Y 439.399,Z 461.751,A -85,B 0,C 180,E1 -8945.34,E2 -8945.34} C_VEL
LIN {X 0,Y 439.392,Z 461.753,A -85,B 0,C 180,E1 -8948.594,E2 -8948.594} C_VEL
LIN {X 0,Y 439.391,Z 461.752,A -85,B 0,C 180,E1 -8951.256,E2 -8951.256} C_VEL
LIN {X 0,Y 439.405,Z 461.75,A -85,B 0,C 180,E1 -8954.729,E2 -8954.729} C_VEL
LIN {X 0,Y 439.401,Z 461.753,A -85,B 0,C 180,E1 -8957.796,E2 -8957.796} C_VEL
LIN {X 0,Y 439.397,Z 461.751,A -85,B 0,C 180,E1 -8960.224,E2 -8960.224} C_VEL
LIN {X 0,Y 439.379,Z 461.755,A -85,B 0,C 180,E1 -8963.713,E2 -8963.713} C_VEL
LIN {X 0,Y 439.374,Z 461.753,A -85,B 0,C 180,E1 -8967.054,E2 -8967.054} C_VEL
LIN {X 0,Y 439.385,Z 461.755,A -85,B 0,C 180,E1 -8970.274,E2 -8970.274} C_VEL
LIN {X 0,Y 439.431,Z 461.748,A -85,B 0,C 180,E1 -8973.396,E2 -8973.396} C_VEL
LIN {X 0,Y 439.388,Z 461.753,A -85,B 0,C 180,E1 -8976.429,E2 -8976.429} C_VEL
LIN {X 0,Y 439.39,Z 461.753,A -85,B 0,C 180,E1 -8979.397,E2 -8979.397} C_VEL
LIN {X 0,Y 439.433,Z 461.746,A -85,B 0,C 180,E1 -8982.309,E2 -8982.309} C_VEL
LIN {X 0,Y 439.449,Z 461.747,A -85,B 0,C 180,E1 -8985.174,E2 -8985.174} C_VEL
LIN {X 0,Y 439.485,Z 461.741,A -85,B 0,C 180,E1 -8988.001,E2 -8988.001} C_VEL
LIN {X 0,Y 439.549,Z 461.734,A -85,B 0,C 180,E1 -8991.726,E2 -8991.726} C_VEL
LIN {X 0,Y 439.622,Z 461.723,A -85,B 0,C 180,E1 -8994.496,E2 -8994.496} C_VEL
LIN {X 0,Y 439.637,Z 461.723,A -85,B 0,C 180,E1 -8998.168,E2 -8998.168} C_VEL
LIN {X 0,Y 439.765,Z 461.708,A -85,B 0,C 180,E1 -9000,E2 -9000} C_VEL
LIN {X 0,Y 439.642,Z 461.719,A -85,B 0,C 180,E1 -9002.749,E2 -9002.749} C_VEL
LIN {X 0,Y 439.619,Z 461.724,A -85,B 0,C 180,E1 -9006.425,E2 -9006.425} C_VEL
LIN {X 0,Y 439.5,Z 461.74,A -85,B 0,C 180,E1 -9009.201,E2 -9009.201} C_VEL
LIN {X 0,Y 439.466,Z 461.745,A -85,B 0,C 180,E1 -9012.937,E2 -9012.937} C_VEL
LIN {X 0,Y 439.448,Z 461.744,A -85,B 0,C 180,E1 -9016.349,E2 -9016.349} C_VEL
LIN {X 0,Y 439.403,Z 461.751,A -85,B 0,C 180,E1 -9019.626,E2 -9019.626} C_VEL
LIN {X 0,Y 439.366,Z 461.756,A -85,B 0,C 180,E1 -9022.575,E2 -9022.575} C_VEL
LIN {X 0,Y 439.406,Z 461.751,A -85,B 0,C 180,E1 -9025.585,E2 -9025.585} C_VEL
LIN {X 0,Y 439.418,Z 461.75,A -85,B 0,C 180,E1 -9028.673,E2 -9028.673} C_VEL
LIN {X 0,Y 439.37,Z 461.753,A -85,B 0,C 180,E1 -9032.03,E2 -9032.03} C_VEL
LIN {X 0,Y 439.396,Z 461.753,A -85,B 0,C 180,E1 -9035.341,E2 -9035.341} C_VEL
LIN {X 0,Y 439.389,Z 461.751,A -85,B 0,C 180,E1 -9038.594,E2 -9038.594} C_VEL
LIN {X 0,Y 439.395,Z 461.753,A -85,B 0,C 180,E1 -9041.258,E2 -9041.258} C_VEL
LIN {X 0,Y 439.407,Z 461.754,A -85,B 0,C 180,E1 -9044.728,E2 -9044.728} C_VEL
LIN {X 0,Y 439.429,Z 461.887,A -85,B 0,C 180,E1 -9048.428,E2 -9048.428} C_VEL
LIN {X 0,Y 440.586,Z 468.353,A -85,B 0,C 180,E1 -9051.53,E2 -9051.53} C_VEL
LIN {X 0,Y 441.351,Z 473.529,A -85,B 0,C 180,E1 -9053.901,E2 -9053.901} C_VEL
LIN {X 0,Y 441.104,Z 478.673,A -85,B 0,C 180,E1 -9056.107,E2 -9056.107} C_VEL
LIN {X 0,Y 440.512,Z 486.832,A -85,B 0,C 180,E1 -9059.488,E2 -9059.488} C_VEL
LIN {X 0,Y 440.055,Z 494.088,A -85,B 0,C 180,E1 -9062.41,E2 -9062.41} C_VEL
LIN {X 0,Y 439.588,Z 502.445,A -85,B 0,C 180,E1 -9065.686,E2 -9065.686} C_VEL
LIN {X 0,Y 439.188,Z 510.816,A -85,B 0,C 180,E1 -9068.897,E2 -9068.897} C_VEL
LIN {X 0,Y 438.928,Z 518.545,A -85,B 0,C 180,E1 -9071.807,E2 -9071.807} C_VEL
LIN {X 0,Y 438.806,Z 523.638,A -85,B 0,C 180,E1 -9073.701,E2 -9073.701} C_VEL
LIN {X 0,Y 440.74,Z 537.339,A -85,B 0,C 180,E1 -9074.184,E2 -9074.184} C_VEL
LIN {X 0,Y 442.042,Z 549.812,A -85,B 0,C 180,E1 -9074.792,E2 -9074.792} C_VEL
LIN {X 0,Y 441.429,Z 561.433,A -85,B 0,C 180,E1 -9075.478,E2 -9075.478} C_VEL
LIN {X 0,Y 440.856,Z 572.842,A -85,B 0,C 180,E1 -9076.339,E2 -9076.339} C_VEL
LIN {X 0,Y 440.275,Z 583.267,A -85,B 0,C 180,E1 -9077.321,E2 -9077.321} C_VEL
LIN {X 0,Y 439.702,Z 593.184,A -85,B 0,C 180,E1 -9078.475,E2 -9078.475} C_VEL
LIN {X 0,Y 439.116,Z 602.836,A -85,B 0,C 180,E1 -9079.86,E2 -9079.86} C_VEL
LIN {X 0,Y 438.81,Z 610.534,A -85,B 0,C 180,E1 -9081.248,E2 -9081.248} C_VEL
LIN {X 0,Y 438.538,Z 616.718,A -85,B 0,C 180,E1 -9082.634,E2 -9082.634} C_VEL
LIN {X 0,Y 438.396,Z 621.445,A -85,B 0,C 180,E1 -9083.965,E2 -9083.965} C_VEL
LIN {X 0,Y 438.358,Z 625.359,A -85,B 0,C 180,E1 -9085.402,E2 -9085.402} C_VEL
LIN {X 0,Y 438.332,Z 627.281,A -85,B 0,C 180,E1 -9086.323,E2 -9086.323} C_VEL
LIN {X 0,Y 438.392,Z 628.749,A -85,B 0,C 180,E1 -9087.244,E2 -9087.244} C_VEL
LIN {X 0,Y 438.366,Z 629.761,A -85,B 0,C 180,E1 -9088.163,E2 -9088.163} C_VEL
LIN {X 0,Y 438.365,Z 630.371,A -85,B 0,C 180,E1 -9089.082,E2 -9089.082} C_VEL
LIN {X 0,Y 438.337,Z 630.577,A -85,B 0,C 180,E1 -9090,E2 -9090} C_VEL
LIN {X 0,Y 438.366,Z 630.34,A -85,B 0,C 180,E1 -9090.919,E2 -9090.919} C_VEL
LIN {X 0,Y 438.368,Z 629.679,A -85,B 0,C 180,E1 -9091.838,E2 -9091.838} C_VEL
LIN {X 0,Y 438.4,Z 628.612,A -85,B 0,C 180,E1 -9092.757,E2 -9092.757} C_VEL
LIN {X 0,Y 438.342,Z 627.124,A -85,B 0,C 180,E1 -9093.677,E2 -9093.677} C_VEL
LIN {X 0,Y 438.422,Z 624.026,A -85,B 0,C 180,E1 -9095.058,E2 -9095.058} C_VEL
LIN {X 0,Y 438.448,Z 619.848,A -85,B 0,C 180,E1 -9096.443,E2 -9096.443} C_VEL
LIN {X 0,Y 438.669,Z 613.449,A -85,B 0,C 180,E1 -9098.059,E2 -9098.059} C_VEL
LIN {X 0,Y 438.956,Z 606.488,A -85,B 0,C 180,E1 -9099.446,E2 -9099.446} C_VEL
LIN {X 0,Y 439.363,Z 597.907,A -85,B 0,C 180,E1 -9100.833,E2 -9100.833} C_VEL
LIN {X 0,Y 439.922,Z 589.133,A -85,B 0,C 180,E1 -9101.987,E2 -9101.987} C_VEL
LIN {X 0,Y 440.435,Z 578.977,A -85,B 0,C 180,E1 -9103.088,E2 -9103.088} C_VEL
LIN {X 0,Y 441.12,Z 567.975,A -85,B 0,C 180,E1 -9104.062,E2 -9104.062} C_VEL
LIN {X 0,Y 441.79,Z 556.693,A -85,B 0,C 180,E1 -9104.864,E2 -9104.864} C_VEL
LIN {X 0,Y 442.068,Z 547.718,A -85,B 0,C 180,E1 -9105.385,E2 -9105.385} C_VEL
LIN {X 0,Y 440.717,Z 533.911,A -85,B 0,C 180,E1 -9106.076,E2 -9106.076} C_VEL
LIN {X 0,Y 438.767,Z 521.127,A -85,B 0,C 180,E1 -9106.594,E2 -9106.594} C_VEL
LIN {X 0,Y 438.983,Z 511.495,A -85,B 0,C 180,E1 -9110.134,E2 -9110.134} C_VEL
LIN {X 0,Y 439.247,Z 503.782,A -85,B 0,C 180,E1 -9113.079,E2 -9113.079} C_VEL
LIN {X 0,Y 439.725,Z 495.084,A -85,B 0,C 180,E1 -9116.585,E2 -9116.585} C_VEL
LIN {X 0,Y 440.209,Z 487.995,A -85,B 0,C 180,E1 -9119.665,E2 -9119.665} C_VEL
LIN {X 0,Y 440.75,Z 482.421,A -85,B 0,C 180,E1 -9122.316,E2 -9122.316} C_VEL
LIN {X 0,Y 441.34,Z 477.408,A -85,B 0,C 180,E1 -9124.979,E2 -9124.979} C_VEL
LIN {X 0,Y 441.447,Z 473.772,A -85,B 0,C 180,E1 -9127.248,E2 -9127.248} C_VEL
LIN {X 0,Y 440.975,Z 470.762,A -85,B 0,C 180,E1 -9129.606,E2 -9129.606} C_VEL
LIN {X 0,Y 440.555,Z 468.312,A -85,B 0,C 180,E1 -9132.068,E2 -9132.068} C_VEL
LIN {X 0,Y 440.223,Z 466.544,A -85,B 0,C 180,E1 -9134.624,E2 -9134.624} C_VEL
LIN {X 0,Y 440.026,Z 465.358,A -85,B 0,C 180,E1 -9137.87,E2 -9137.87} C_VEL
LIN {X 0,Y 439.94,Z 465.184,A -85,B 0,C 180,E1 -9140.283,E2 -9140.283} C_VEL
LIN {X 0,Y 439.95,Z 465.547,A -85,B 0,C 180,E1 -9143.009,E2 -9143.009} C_VEL
LIN {X 0,Y 439.922,Z 466.128,A -85,B 0,C 180,E1 -9144.892,E2 -9144.892} C_VEL
LIN {X 0,Y 439.676,Z 467.615,A -85,B 0,C 180,E1 -9148.164,E2 -9148.164} C_VEL
LIN {X 0,Y 439.383,Z 469.659,A -85,B 0,C 180,E1 -9151.611,E2 -9151.611} C_VEL
LIN {X 0,Y 439.159,Z 471.579,A -85,B 0,C 180,E1 -9154.4,E2 -9154.4} C_VEL
LIN {X 0,Y 438.986,Z 473.84,A -85,B 0,C 180,E1 -9157.404,E2 -9157.404} C_VEL
LIN {X 0,Y 438.856,Z 476.233,A -85,B 0,C 180,E1 -9160.348,E2 -9160.348} C_VEL
LIN {X 0,Y 438.8,Z 479.014,A -85,B 0,C 180,E1 -9163.564,E2 -9163.564} C_VEL
LIN {X 0,Y 442.176,Z 491.192,A -85,B 0,C 180,E1 -9164.187,E2 -9164.187} C_VEL
LIN {X 0,Y 443.054,Z 496.364,A -85,B 0,C 180,E1 -9164.474,E2 -9164.474} C_VEL
LIN {X 0,Y 442.518,Z 508.604,A -85,B 0,C 180,E1 -9165.162,E2 -9165.162} C_VEL
LIN {X 0,Y 441.863,Z 520.909,A -85,B 0,C 180,E1 -9166.062,E2 -9166.062} C_VEL
LIN {X 0,Y 441.22,Z 532.255,A -85,B 0,C 180,E1 -9167.115,E2 -9167.115} C_VEL
LIN {X 0,Y 440.547,Z 542.238,A -85,B 0,C 180,E1 -9168.264,E2 -9168.264} C_VEL
LIN {X 0,Y 439.943,Z 551.84,A -85,B 0,C 180,E1 -9169.647,E2 -9169.647} C_VEL
LIN {X 0,Y 439.481,Z 559.568,A -85,B 0,C 180,E1 -9171.03,E2 -9171.03} C_VEL
LIN {X 0,Y 439.157,Z 564.797,A -85,B 0,C 180,E1 -9172.182,E2 -9172.182} C_VEL
LIN {X 0,Y 438.906,Z 569.893,A -85,B 0,C 180,E1 -9173.564,E2 -9173.564} C_VEL
LIN {X 0,Y 438.658,Z 573.844,A -85,B 0,C 180,E1 -9174.945,E2 -9174.945} C_VEL
LIN {X 0,Y 438.568,Z 576.739,A -85,B 0,C 180,E1 -9176.325,E2 -9176.325} C_VEL
LIN {X 0,Y 438.497,Z 578.115,A -85,B 0,C 180,E1 -9177.244,E2 -9177.244} C_VEL
LIN {X 0,Y 438.465,Z 579.07,A -85,B 0,C 180,E1 -9178.163,E2 -9178.163} C_VEL
LIN {X 0,Y 438.368,Z 579.638,A -85,B 0,C 180,E1 -9179.082,E2 -9179.082} C_VEL
LIN {X 0,Y 438.339,Z 579.807,A -85,B 0,C 180,E1 -9180,E2 -9180} C_VEL
LIN {X 0,Y 438.368,Z 579.531,A -85,B 0,C 180,E1 -9180.919,E2 -9180.919} C_VEL
LIN {X 0,Y 438.417,Z 578.858,A -85,B 0,C 180,E1 -9181.837,E2 -9181.837} C_VEL
LIN {X 0,Y 438.473,Z 577.791,A -85,B 0,C 180,E1 -9182.756,E2 -9182.756} C_VEL
LIN {X 0,Y 438.55,Z 576.305,A -85,B 0,C 180,E1 -9183.676,E2 -9183.676} C_VEL
LIN {X 0,Y 438.55,Z 573.247,A -85,B 0,C 180,E1 -9185.057,E2 -9185.057} C_VEL
LIN {X 0,Y 438.843,Z 569.115,A -85,B 0,C 180,E1 -9186.437,E2 -9186.437} C_VEL
LIN {X 0,Y 439.061,Z 562.782,A -85,B 0,C 180,E1 -9188.052,E2 -9188.052} C_VEL
LIN {X 0,Y 439.463,Z 555.889,A -85,B 0,C 180,E1 -9189.435,E2 -9189.435} C_VEL
LIN {X 0,Y 439.839,Z 548.87,A -85,B 0,C 180,E1 -9190.589,E2 -9190.589} C_VEL
LIN {X 0,Y 440.275,Z 540.435,A -85,B 0,C 180,E1 -9191.743,E2 -9191.743} C_VEL
LIN {X 0,Y 440.959,Z 530.059,A -85,B 0,C 180,E1 -9192.893,E2 -9192.893} C_VEL
LIN {X 0,Y 441.463,Z 518.456,A -85,B 0,C 180,E1 -9193.933,E2 -9193.933} C_VEL
LIN {X 0,Y 441.995,Z 507.041,A -85,B 0,C 180,E1 -9194.739,E2 -9194.739} C_VEL
LIN {X 0,Y 442.481,Z 495.475,A -85,B 0,C 180,E1 -9195.37,E2 -9195.37} C_VEL
LIN {X 0,Y 441.325,Z 488.815,A -85,B 0,C 180,E1 -9195.708,E2 -9195.708} C_VEL
LIN {X 0,Y 438.493,Z 476.161,A -85,B 0,C 180,E1 -9196.254,E2 -9196.254} C_VEL
LIN {X 0,Y 438.499,Z 472.466,A -85,B 0,C 180,E1 -9199.669,E2 -9199.669} C_VEL
LIN {X 0,Y 438.542,Z 469.335,A -85,B 0,C 180,E1 -9202.621,E2 -9202.621} C_VEL
LIN {X 0,Y 438.665,Z 465.591,A -85,B 0,C 180,E1 -9206.208,E2 -9206.208} C_VEL
LIN {X 0,Y 438.668,Z 463.017,A -85,B 0,C 180,E1 -9208.727,E2 -9208.727} C_VEL
LIN {X 0,Y 438.729,Z 461.839,A -85,B 0,C 180,E1 -9210.114,E2 -9210.114} C_VEL
LIN {X 0,Y 439.044,Z 461.797,A -85,B 0,C 180,E1 -9212.974,E2 -9212.974} C_VEL
LIN {X 0,Y 439.309,Z 461.763,A -85,B 0,C 180,E1 -9215.324,E2 -9215.324} C_VEL
LIN {X 0,Y 439.382,Z 461.754,A -85,B 0,C 180,E1 -9218.596,E2 -9218.596} C_VEL
LIN {X 0,Y 439.393,Z 461.752,A -85,B 0,C 180,E1 -9221.257,E2 -9221.257} C_VEL
LIN {X 0,Y 439.404,Z 461.751,A -85,B 0,C 180,E1 -9224.73,E2 -9224.73} C_VEL
LIN {X 0,Y 439.401,Z 461.753,A -85,B 0,C 180,E1 -9227.796,E2 -9227.796} C_VEL
LIN {X 0,Y 439.435,Z 461.748,A -85,B 0,C 180,E1 -9230.228,E2 -9230.228} C_VEL
LIN {X 0,Y 439.379,Z 461.754,A -85,B 0,C 180,E1 -9233.713,E2 -9233.713} C_VEL
LIN {X 0,Y 439.378,Z 461.754,A -85,B 0,C 180,E1 -9237.054,E2 -9237.054} C_VEL
LIN {X 0,Y 439.387,Z 461.756,A -85,B 0,C 180,E1 -9240.274,E2 -9240.274} C_VEL
LIN {X 0,Y 439.434,Z 461.748,A -85,B 0,C 180,E1 -9243.396,E2 -9243.396} C_VEL
LIN {X 0,Y 439.393,Z 461.754,A -85,B 0,C 180,E1 -9246.43,E2 -9246.43} C_VEL
LIN {X 0,Y 439.394,Z 461.752,A -85,B 0,C 180,E1 -9249.397,E2 -9249.397} C_VEL
LIN {X 0,Y 439.436,Z 461.749,A -85,B 0,C 180,E1 -9252.309,E2 -9252.309} C_VEL
LIN {X 0,Y 439.454,Z 461.742,A -85,B 0,C 180,E1 -9255.174,E2 -9255.174} C_VEL
LIN {X 0,Y 439.489,Z 461.741,A -85,B 0,C 180,E1 -9258.001,E2 -9258.001} C_VEL
LIN {X 0,Y 439.537,Z 461.735,A -85,B 0,C 180,E1 -9261.726,E2 -9261.726} C_VEL
LIN {X 0,Y 439.625,Z 461.724,A -85,B 0,C 180,E1 -9264.496,E2 -9264.496} C_VEL
LIN {X 0,Y 439.573,Z 461.729,A -85,B 0,C 180,E1 -9266.989,E2 -9266.989} C_VEL
LIN {X 0,Y 439.049,Z 461.797,A -85,B 0,C 180,E1 -9267.754,E2 -9267.754} C_VEL
LIN {X 0,Y 436.232,Z 462.148,A -85,B 0,C 180,E1 -9268.997,E2 -9268.997} C_VEL
LIN {X 0,Y 433.755,Z 462.457,A -85,B 0,C 180,E1 -9270,E2 -9270} C_VEL
LIN {X 0,Y 432.676,Z 462.589,A -85,B 0,C 180,E1 -9270.776,E2 -9270.776} C_VEL
LIN {X 0,Y 432.585,Z 462.599,A -85,B 0,C 180,E1 -9271.039,E2 -9271.039} C_VEL
LIN {X 0,Y 432.597,Z 462.599,A -85,B 0,C 180,E1 -9272.793,E2 -9272.793} C_VEL
LIN {X 0,Y 432.591,Z 462.6,A -85,B 0,C 180,E1 -9275.594,E2 -9275.594} C_VEL
LIN {X 0,Y 432.488,Z 462.613,A -85,B 0,C 180,E1 -9278.41,E2 -9278.41} C_VEL
LIN {X 0,Y 432.465,Z 462.618,A -85,B 0,C 180,E1 -9282.196,E2 -9282.196} C_VEL
LIN {X 0,Y 432.436,Z 462.62,A -85,B 0,C 180,E1 -9286.038,E2 -9286.038} C_VEL
LIN {X 0,Y 432.392,Z 462.624,A -85,B 0,C 180,E1 -9289.485,E2 -9289.485} C_VEL
LIN {X 0,Y 432.324,Z 462.632,A -85,B 0,C 180,E1 -9292.964,E2 -9292.964} C_VEL
LIN {X 0,Y 432.369,Z 462.63,A -85,B 0,C 180,E1 -9296.032,E2 -9296.032} C_VEL
LIN {X 0,Y 432.347,Z 462.629,A -85,B 0,C 180,E1 -9299.187,E2 -9299.187} C_VEL
LIN {X 0,Y 432.327,Z 462.633,A -85,B 0,C 180,E1 -9302.443,E2 -9302.443} C_VEL
LIN {X 0,Y 432.349,Z 462.632,A -85,B 0,C 180,E1 -9305.632,E2 -9305.632} C_VEL
LIN {X 0,Y 432.354,Z 462.629,A -85,B 0,C 180,E1 -9308.716,E2 -9308.716} C_VEL
LIN {X 0,Y 432.337,Z 462.634,A -85,B 0,C 180,E1 -9311.797,E2 -9311.797} C_VEL
LIN {X 0,Y 432.336,Z 462.631,A -85,B 0,C 180,E1 -9314.347,E2 -9314.347} C_VEL
LIN {X 0,Y 432.327,Z 462.633,A -85,B 0,C 180,E1 -9317.015,E2 -9317.015} C_VEL
LIN {X 0,Y 432.336,Z 462.634,A -85,B 0,C 180,E1 -9319.82,E2 -9319.82} C_VEL
LIN {X 0,Y 432.317,Z 462.634,A -85,B 0,C 180,E1 -9323.023,E2 -9323.023} C_VEL
LIN {X 0,Y 432.362,Z 462.63,A -85,B 0,C 180,E1 -9325.996,E2 -9325.996} C_VEL
LIN {X 0,Y 432.349,Z 462.632,A -85,B 0,C 180,E1 -9329.489,E2 -9329.489} C_VEL
LIN {X 0,Y 432.394,Z 462.623,A -85,B 0,C 180,E1 -9332.928,E2 -9332.928} C_VEL
LIN {X 0,Y 432.373,Z 462.627,A -85,B 0,C 180,E1 -9336.023,E2 -9336.023} C_VEL
LIN {X 0,Y 432.352,Z 462.63,A -85,B 0,C 180,E1 -9339.046,E2 -9339.046} C_VEL
LIN {X 0,Y 432.38,Z 462.626,A -85,B 0,C 180,E1 -9342.011,E2 -9342.011} C_VEL
LIN {X 0,Y 432.397,Z 462.625,A -85,B 0,C 180,E1 -9344.926,E2 -9344.926} C_VEL
LIN {X 0,Y 432.461,Z 462.618,A -85,B 0,C 180,E1 -9347.803,E2 -9347.803} C_VEL
LIN {X 0,Y 432.493,Z 462.613,A -85,B 0,C 180,E1 -9351.59,E2 -9351.59} C_VEL
LIN {X 0,Y 432.599,Z 462.597,A -85,B 0,C 180,E1 -9354.406,E2 -9354.406} C_VEL
LIN {X 0,Y 432.607,Z 462.598,A -85,B 0,C 180,E1 -9358.138,E2 -9358.138} C_VEL
LIN {X 0,Y 432.735,Z 462.583,A -85,B 0,C 180,E1 -9360,E2 -9360} C_VEL
LIN {X 0,Y 432.593,Z 462.598,A -85,B 0,C 180,E1 -9362.793,E2 -9362.793} C_VEL
LIN {X 0,Y 432.574,Z 462.602,A -85,B 0,C 180,E1 -9366.53,E2 -9366.53} C_VEL
LIN {X 0,Y 432.443,Z 462.62,A -85,B 0,C 180,E1 -9369.353,E2 -9369.353} C_VEL
LIN {X 0,Y 432.431,Z 462.62,A -85,B 0,C 180,E1 -9372.803,E2 -9372.803} C_VEL
LIN {X 0,Y 432.413,Z 462.62,A -85,B 0,C 180,E1 -9376.479,E2 -9376.479} C_VEL
LIN {X 0,Y 432.34,Z 462.632,A -85,B 0,C 180,E1 -9379.96,E2 -9379.96} C_VEL
LIN {X 0,Y 432.32,Z 462.633,A -85,B 0,C 180,E1 -9382.964,E2 -9382.964} C_VEL
LIN {X 0,Y 432.365,Z 462.627,A -85,B 0,C 180,E1 -9386.032,E2 -9386.032} C_VEL
LIN {X 0,Y 432.343,Z 462.631,A -85,B 0,C 180,E1 -9389.187,E2 -9389.187} C_VEL
LIN {X 0,Y 432.323,Z 462.631,A -85,B 0,C 180,E1 -9392.443,E2 -9392.443} C_VEL
LIN {X 0,Y 432.346,Z 462.632,A -85,B 0,C 180,E1 -9395.632,E2 -9395.632} C_VEL
LIN {X 0,Y 432.351,Z 462.628,A -85,B 0,C 180,E1 -9398.716,E2 -9398.716} C_VEL
LIN {X 0,Y 432.371,Z 462.628,A -85,B 0,C 180,E1 -9401.793,E2 -9401.793} C_VEL
LIN {X 0,Y 432.379,Z 462.63,A -85,B 0,C 180,E1 -9404.342,E2 -9404.342} C_VEL
LIN {X 0,Y 432.372,Z 462.681,A -85,B 0,C 180,E1 -9408.13,E2 -9408.13} C_VEL
LIN {X 0,Y 433.452,Z 468.754,A -85,B 0,C 180,E1 -9411.103,E2 -9411.103} C_VEL
LIN {X 0,Y 434.201,Z 473.24,A -85,B 0,C 180,E1 -9413.21,E2 -9413.21} C_VEL
LIN {X 0,Y 434.298,Z 477.093,A -85,B 0,C 180,E1 -9414.937,E2 -9414.937} C_VEL
LIN {X 0,Y 433.666,Z 484.794,A -85,B 0,C 180,E1 -9418.218,E2 -9418.218} C_VEL
LIN {X 0,Y 433.229,Z 491.902,A -85,B 0,C 180,E1 -9421.165,E2 -9421.165} C_VEL
LIN {X 0,Y 432.674,Z 500.182,A -85,B 0,C 180,E1 -9424.504,E2 -9424.504} C_VEL
LIN {X 0,Y 432.208,Z 508.95,A -85,B 0,C 180,E1 -9427.951,E2 -9427.951} C_VEL
LIN {X 0,Y 431.861,Z 518.156,A -85,B 0,C 180,E1 -9431.498,E2 -9431.498} C_VEL
LIN {X 0,Y 431.74,Z 523.29,A -85,B 0,C 180,E1 -9433.452,E2 -9433.452} C_VEL
LIN {X 0,Y 433.835,Z 538.3,A -85,B 0,C 180,E1 -9434.015,E2 -9434.015} C_VEL
LIN {X 0,Y 435.095,Z 549.909,A -85,B 0,C 180,E1 -9434.603,E2 -9434.603} C_VEL
LIN {X 0,Y 434.418,Z 562.259,A -85,B 0,C 180,E1 -9435.358,E2 -9435.358} C_VEL
LIN {X 0,Y 433.793,Z 573.817,A -85,B 0,C 180,E1 -9436.269,E2 -9436.269} C_VEL
LIN {X 0,Y 433.15,Z 584.688,A -85,B 0,C 180,E1 -9437.347,E2 -9437.347} C_VEL
LIN {X 0,Y 432.587,Z 594.31,A -85,B 0,C 180,E1 -9438.521,E2 -9438.521} C_VEL
LIN {X 0,Y 432.076,Z 602.226,A -85,B 0,C 180,E1 -9439.693,E2 -9439.693} C_VEL
LIN {X 0,Y 431.724,Z 609.975,A -85,B 0,C 180,E1 -9441.104,E2 -9441.104} C_VEL
LIN {X 0,Y 431.465,Z 616.193,A -85,B 0,C 180,E1 -9442.513,E2 -9442.513} C_VEL
LIN {X 0,Y 431.299,Z 621.369,A -85,B 0,C 180,E1 -9444.002,E2 -9444.002} C_VEL
LIN {X 0,Y 431.289,Z 624.889,A -85,B 0,C 180,E1 -9445.327,E2 -9445.327} C_VEL
LIN {X 0,Y 431.238,Z 626.819,A -85,B 0,C 180,E1 -9446.262,E2 -9446.262} C_VEL
LIN {X 0,Y 431.318,Z 628.308,A -85,B 0,C 180,E1 -9447.198,E2 -9447.198} C_VEL
LIN {X 0,Y 431.285,Z 629.327,A -85,B 0,C 180,E1 -9448.133,E2 -9448.133} C_VEL
LIN {X 0,Y 431.289,Z 629.944,A -85,B 0,C 180,E1 -9449.067,E2 -9449.067} C_VEL
LIN {X 0,Y 431.277,Z 630.156,A -85,B 0,C 180,E1 -9450,E2 -9450} C_VEL
LIN {X 0,Y 431.276,Z 629.931,A -85,B 0,C 180,E1 -9450.934,E2 -9450.934} C_VEL
LIN {X 0,Y 431.287,Z 629.272,A -85,B 0,C 180,E1 -9451.868,E2 -9451.868} C_VEL
LIN {X 0,Y 431.326,Z 628.209,A -85,B 0,C 180,E1 -9452.802,E2 -9452.802} C_VEL
LIN {X 0,Y 431.245,Z 626.724,A -85,B 0,C 180,E1 -9453.738,E2 -9453.738} C_VEL
LIN {X 0,Y 431.329,Z 623.63,A -85,B 0,C 180,E1 -9455.142,E2 -9455.142} C_VEL
LIN {X 0,Y 431.376,Z 619.458,A -85,B 0,C 180,E1 -9456.549,E2 -9456.549} C_VEL
LIN {X 0,Y 431.601,Z 613.078,A -85,B 0,C 180,E1 -9458.192,E2 -9458.192} C_VEL
LIN {X 0,Y 431.892,Z 606.138,A -85,B 0,C 180,E1 -9459.602,E2 -9459.602} C_VEL
LIN {X 0,Y 432.365,Z 597.584,A -85,B 0,C 180,E1 -9461.011,E2 -9461.011} C_VEL
LIN {X 0,Y 432.9,Z 588.863,A -85,B 0,C 180,E1 -9462.184,E2 -9462.184} C_VEL
LIN {X 0,Y 433.491,Z 578.873,A -85,B 0,C 180,E1 -9463.292,E2 -9463.292} C_VEL
LIN {X 0,Y 434.224,Z 567.867,A -85,B 0,C 180,E1 -9464.29,E2 -9464.29} C_VEL
LIN {X 0,Y 434.931,Z 556.769,A -85,B 0,C 180,E1 -9465.104,E2 -9465.104} C_VEL
LIN {X 0,Y 435.128,Z 547.969,A -85,B 0,C 180,E1 -9465.636,E2 -9465.636} C_VEL
LIN {X 0,Y 433.873,Z 534.193,A -85,B 0,C 180,E1 -9466.359,E2 -9466.359} C_VEL
LIN {X 0,Y 431.664,Z 520.58,A -85,B 0,C 180,E1 -9466.942,E2 -9466.942} C_VEL
LIN {X 0,Y 431.957,Z 511.211,A -85,B 0,C 180,E1 -9470.476,E2 -9470.476} C_VEL
LIN {X 0,Y 432.235,Z 503.577,A -85,B 0,C 180,E1 -9473.476,E2 -9473.476} C_VEL
LIN {X 0,Y 432.696,Z 495.78,A -85,B 0,C 180,E1 -9476.705,E2 -9476.705} C_VEL
LIN {X 0,Y 433.191,Z 489.162,A -85,B 0,C 180,E1 -9479.659,E2 -9479.659} C_VEL
LIN {X 0,Y 433.75,Z 483.692,A -85,B 0,C 180,E1 -9482.324,E2 -9482.324} C_VEL
LIN {X 0,Y 434.281,Z 479.633,A -85,B 0,C 180,E1 -9484.5,E2 -9484.5} C_VEL
LIN {X 0,Y 434.483,Z 475.963,A -85,B 0,C 180,E1 -9486.763,E2 -9486.763} C_VEL
LIN {X 0,Y 434.141,Z 472.803,A -85,B 0,C 180,E1 -9489.15,E2 -9489.15} C_VEL
LIN {X 0,Y 433.677,Z 470.093,A -85,B 0,C 180,E1 -9491.801,E2 -9491.801} C_VEL
LIN {X 0,Y 433.308,Z 468.189,A -85,B 0,C 180,E1 -9494.467,E2 -9494.467} C_VEL
LIN {X 0,Y 433.135,Z 467.082,A -85,B 0,C 180,E1 -9497.04,E2 -9497.04} C_VEL
LIN {X 0,Y 432.999,Z 466.648,A -85,B 0,C 180,E1 -9499.717,E2 -9499.717} C_VEL
LIN {X 0,Y 432.988,Z 466.95,A -85,B 0,C 180,E1 -9503.09,E2 -9503.09} C_VEL
LIN {X 0,Y 432.852,Z 467.822,A -85,B 0,C 180,E1 -9505.901,E2 -9505.901} C_VEL
LIN {X 0,Y 432.638,Z 469.107,A -85,B 0,C 180,E1 -9508.68,E2 -9508.68} C_VEL
LIN {X 0,Y 432.334,Z 470.951,A -85,B 0,C 180,E1 -9511.873,E2 -9511.873} C_VEL
LIN {X 0,Y 432.116,Z 473.054,A -85,B 0,C 180,E1 -9514.984,E2 -9514.984} C_VEL
LIN {X 0,Y 431.943,Z 475.335,A -85,B 0,C 180,E1 -9518.038,E2 -9518.038} C_VEL
LIN {X 0,Y 431.87,Z 477.718,A -85,B 0,C 180,E1 -9521.006,E2 -9521.006} C_VEL
LIN {X 0,Y 431.796,Z 479.791,A -85,B 0,C 180,E1 -9523.228,E2 -9523.228} C_VEL
LIN {X 0,Y 435.364,Z 492.152,A -85,B 0,C 180,E1 -9523.9,E2 -9523.9} C_VEL
LIN {X 0,Y 436.317,Z 497.847,A -85,B 0,C 180,E1 -9524.228,E2 -9524.228} C_VEL
LIN {X 0,Y 435.766,Z 509.831,A -85,B 0,C 180,E1 -9524.926,E2 -9524.926} C_VEL
LIN {X 0,Y 435.054,Z 521.851,A -85,B 0,C 180,E1 -9525.834,E2 -9525.834} C_VEL
LIN {X 0,Y 434.349,Z 533.083,A -85,B 0,C 180,E1 -9526.907,E2 -9526.907} C_VEL
LIN {X 0,Y 433.634,Z 542.93,A -85,B 0,C 180,E1 -9528.075,E2 -9528.075} C_VEL
LIN {X 0,Y 432.986,Z 552.482,A -85,B 0,C 180,E1 -9529.479,E2 -9529.479} C_VEL
LIN {X 0,Y 432.503,Z 560.172,A -85,B 0,C 180,E1 -9530.884,E2 -9530.884} C_VEL
LIN {X 0,Y 432.004,Z 567.193,A -85,B 0,C 180,E1 -9532.522,E2 -9532.522} C_VEL
LIN {X 0,Y 431.741,Z 571.862,A -85,B 0,C 180,E1 -9533.926,E2 -9533.926} C_VEL
LIN {X 0,Y 431.63,Z 575.41,A -85,B 0,C 180,E1 -9535.33,E2 -9535.33} C_VEL
LIN {X 0,Y 431.516,Z 577.232,A -85,B 0,C 180,E1 -9536.265,E2 -9536.265} C_VEL
LIN {X 0,Y 431.425,Z 578.584,A -85,B 0,C 180,E1 -9537.199,E2 -9537.199} C_VEL
LIN {X 0,Y 431.41,Z 579.522,A -85,B 0,C 180,E1 -9538.133,E2 -9538.133} C_VEL
LIN {X 0,Y 431.31,Z 580.076,A -85,B 0,C 180,E1 -9539.067,E2 -9539.067} C_VEL
LIN {X 0,Y 431.278,Z 580.227,A -85,B 0,C 180,E1 -9540,E2 -9540} C_VEL
LIN {X 0,Y 431.293,Z 579.934,A -85,B 0,C 180,E1 -9540.934,E2 -9540.934} C_VEL
LIN {X 0,Y 431.334,Z 579.244,A -85,B 0,C 180,E1 -9541.868,E2 -9541.868} C_VEL
LIN {X 0,Y 431.403,Z 578.161,A -85,B 0,C 180,E1 -9542.802,E2 -9542.802} C_VEL
LIN {X 0,Y 431.474,Z 576.648,A -85,B 0,C 180,E1 -9543.736,E2 -9543.736} C_VEL
LIN {X 0,Y 431.485,Z 573.556,A -85,B 0,C 180,E1 -9545.14,E2 -9545.14} C_VEL
LIN {X 0,Y 431.785,Z 569.382,A -85,B 0,C 180,E1 -9546.543,E2 -9546.543} C_VEL
LIN {X 0,Y 432.011,Z 562.998,A -85,B 0,C 180,E1 -9548.184,E2 -9548.184} C_VEL
LIN {X 0,Y 432.455,Z 556.058,A -85,B 0,C 180,E1 -9549.589,E2 -9549.589} C_VEL
LIN {X 0,Y 432.86,Z 548.987,A -85,B 0,C 180,E1 -9550.762,E2 -9550.762} C_VEL
LIN {X 0,Y 433.304,Z 540.485,A -85,B 0,C 180,E1 -9551.935,E2 -9551.935} C_VEL
LIN {X 0,Y 434.032,Z 530.023,A -85,B 0,C 180,E1 -9553.103,E2 -9553.103} C_VEL
LIN {X 0,Y 434.569,Z 518.342,A -85,B 0,C 180,E1 -9554.159,E2 -9554.159} C_VEL
LIN {X 0,Y 435.138,Z 506.769,A -85,B 0,C 180,E1 -9554.977,E2 -9554.977} C_VEL
LIN {X 0,Y 435.504,Z 495.064,A -85,B 0,C 180,E1 -9555.623,E2 -9555.623} C_VEL
LIN {X 0,Y 432.548,Z 481.624,A -85,B 0,C 180,E1 -9556.281,E2 -9556.281} C_VEL
LIN {X 0,Y 431.414,Z 476.484,A -85,B 0,C 180,E1 -9556.504,E2 -9556.504} C_VEL
LIN {X 0,Y 431.42,Z 472.725,A -85,B 0,C 180,E1 -9560.005,E2 -9560.005} C_VEL
LIN {X 0,Y 431.498,Z 469.551,A -85,B 0,C 180,E1 -9563.011,E2 -9563.011} C_VEL
LIN {X 0,Y 431.602,Z 466.032,A -85,B 0,C 180,E1 -9566.415,E2 -9566.415} C_VEL
LIN {X 0,Y 431.614,Z 463.164,A -85,B 0,C 180,E1 -9569.242,E2 -9569.242} C_VEL
LIN {X 0,Y 431.704,Z 462.713,A -85,B 0,C 180,E1 -9570.364,E2 -9570.364} C_VEL
LIN {X 0,Y 432.06,Z 462.666,A -85,B 0,C 180,E1 -9573.577,E2 -9573.577} C_VEL
LIN {X 0,Y 432.26,Z 462.642,A -85,B 0,C 180,E1 -9575.826,E2 -9575.826} C_VEL
LIN {X 0,Y 432.346,Z 462.63,A -85,B 0,C 180,E1 -9578.715,E2 -9578.715} C_VEL
LIN {X 0,Y 432.338,Z 462.633,A -85,B 0,C 180,E1 -9581.797,E2 -9581.797} C_VEL
LIN {X 0,Y 432.338,Z 462.634,A -85,B 0,C 180,E1 -9584.347,E2 -9584.347} C_VEL
LIN {X 0,Y 432.325,Z 462.632,A -85,B 0,C 180,E1 -9587.016,E2 -9587.016} C_VEL
LIN {X 0,Y 432.341,Z 462.632,A -85,B 0,C 180,E1 -9589.82,E2 -9589.82} C_VEL
LIN {X 0,Y 432.315,Z 462.631,A -85,B 0,C 180,E1 -9593.023,E2 -9593.023} C_VEL
LIN {X 0,Y 432.364,Z 462.629,A -85,B 0,C 180,E1 -9595.997,E2 -9595.997} C_VEL
LIN {X 0,Y 432.352,Z 462.628,A -85,B 0,C 180,E1 -9599.49,E2 -9599.49} C_VEL
LIN {X 0,Y 432.396,Z 462.624,A -85,B 0,C 180,E1 -9602.928,E2 -9602.928} C_VEL
LIN {X 0,Y 432.377,Z 462.627,A -85,B 0,C 180,E1 -9606.023,E2 -9606.023} C_VEL
LIN {X 0,Y 432.356,Z 462.628,A -85,B 0,C 180,E1 -9609.046,E2 -9609.046} C_VEL
LIN {X 0,Y 432.383,Z 462.626,A -85,B 0,C 180,E1 -9612.011,E2 -9612.011} C_VEL
LIN {X 0,Y 432.401,Z 462.621,A -85,B 0,C 180,E1 -9614.926,E2 -9614.926} C_VEL
LIN {X 0,Y 432.465,Z 462.617,A -85,B 0,C 180,E1 -9617.803,E2 -9617.803} C_VEL
LIN {X 0,Y 432.487,Z 462.612,A -85,B 0,C 180,E1 -9621.59,E2 -9621.59} C_VEL
LIN {X 0,Y 432.601,Z 462.599,A -85,B 0,C 180,E1 -9624.406,E2 -9624.406} C_VEL
LIN {X 0,Y 432.61,Z 462.601,A -85,B 0,C 180,E1 -9628.138,E2 -9628.138} C_VEL
LIN {X 0,Y 432.738,Z 462.584,A -85,B 0,C 180,E1 -9630,E2 -9630} C_VEL
LIN {X 0,Y 432.585,Z 462.599,A -85,B 0,C 180,E1 -9631.039,E2 -9631.039} C_VEL
LIN {X 0,Y 431.879,Z 462.69,A -85,B 0,C 180,E1 -9631.815,E2 -9631.815} C_VEL
LIN {X 0,Y 428.909,Z 463.058,A -85,B 0,C 180,E1 -9633.075,E2 -9633.075} C_VEL
LIN {X 0,Y 426.455,Z 463.366,A -85,B 0,C 180,E1 -9634.091,E2 -9634.091} C_VEL
LIN {X 0,Y 425.473,Z 463.485,A -85,B 0,C 180,E1 -9634.879,E2 -9634.879} C_VEL
LIN {X 0,Y 425.431,Z 463.489,A -85,B 0,C 180,E1 -9635.145,E2 -9635.145} C_VEL
LIN {X 0,Y 425.484,Z 463.487,A -85,B 0,C 180,E1 -9637.663,E2 -9637.663} C_VEL
LIN {X 0,Y 425.372,Z 463.5,A -85,B 0,C 180,E1 -9640.471,E2 -9640.471} C_VEL
LIN {X 0,Y 425.37,Z 463.498,A -85,B 0,C 180,E1 -9643.374,E2 -9643.374} C_VEL
LIN {X 0,Y 425.366,Z 463.5,A -85,B 0,C 180,E1 -9646.605,E2 -9646.605} C_VEL
LIN {X 0,Y 425.333,Z 463.504,A -85,B 0,C 180,E1 -9649.635,E2 -9649.635} C_VEL
LIN {X 0,Y 425.311,Z 463.507,A -85,B 0,C 180,E1 -9653.365,E2 -9653.365} C_VEL
LIN {X 0,Y 425.351,Z 463.5,A -85,B 0,C 180,E1 -9656.844,E2 -9656.844} C_VEL
LIN {X 0,Y 425.295,Z 463.511,A -85,B 0,C 180,E1 -9659.719,E2 -9659.719} C_VEL
LIN {X 0,Y 425.286,Z 463.509,A -85,B 0,C 180,E1 -9663.048,E2 -9663.048} C_VEL
LIN {X 0,Y 425.288,Z 463.511,A -85,B 0,C 180,E1 -9665.929,E2 -9665.929} C_VEL
LIN {X 0,Y 425.303,Z 463.508,A -85,B 0,C 180,E1 -9669.043,E2 -9669.043} C_VEL
LIN {X 0,Y 425.279,Z 463.508,A -85,B 0,C 180,E1 -9672.652,E2 -9672.652} C_VEL
LIN {X 0,Y 425.271,Z 463.513,A -85,B 0,C 180,E1 -9676.045,E2 -9676.045} C_VEL
LIN {X 0,Y 425.278,Z 463.509,A -85,B 0,C 180,E1 -9678.621,E2 -9678.621} C_VEL
LIN {X 0,Y 425.302,Z 463.507,A -85,B 0,C 180,E1 -9681.101,E2 -9681.101} C_VEL
LIN {X 0,Y 425.303,Z 463.507,A -85,B 0,C 180,E1 -9684.664,E2 -9684.664} C_VEL
LIN {X 0,Y 425.267,Z 463.512,A -85,B 0,C 180,E1 -9688.073,E2 -9688.073} C_VEL
LIN {X 0,Y 425.333,Z 463.504,A -85,B 0,C 180,E1 -9691.368,E2 -9691.368} C_VEL
LIN {X 0,Y 425.297,Z 463.506,A -85,B 0,C 180,E1 -9694.554,E2 -9694.554} C_VEL
LIN {X 0,Y 425.289,Z 463.51,A -85,B 0,C 180,E1 -9697.661,E2 -9697.661} C_VEL
LIN {X 0,Y 425.364,Z 463.498,A -85,B 0,C 180,E1 -9700.704,E2 -9700.704} C_VEL
LIN {X 0,Y 425.39,Z 463.498,A -85,B 0,C 180,E1 -9703.688,E2 -9703.688} C_VEL
LIN {X 0,Y 425.413,Z 463.496,A -85,B 0,C 180,E1 -9707.598,E2 -9707.598} C_VEL
LIN {X 0,Y 425.444,Z 463.491,A -85,B 0,C 180,E1 -9711.45,E2 -9711.45} C_VEL
LIN {X 0,Y 425.555,Z 463.475,A -85,B 0,C 180,E1 -9714.313,E2 -9714.313} C_VEL
LIN {X 0,Y 425.577,Z 463.474,A -85,B 0,C 180,E1 -9718.107,E2 -9718.107} C_VEL
LIN {X 0,Y 425.705,Z 463.459,A -85,B 0,C 180,E1 -9720,E2 -9720} C_VEL
LIN {X 0,Y 425.547,Z 463.475,A -85,B 0,C 180,E1 -9722.84,E2 -9722.84} C_VEL
LIN {X 0,Y 425.532,Z 463.479,A -85,B 0,C 180,E1 -9726.639,E2 -9726.639} C_VEL
LIN {X 0,Y 425.401,Z 463.498,A -85,B 0,C 180,E1 -9729.509,E2 -9729.509} C_VEL
LIN {X 0,Y 425.394,Z 463.497,A -85,B 0,C 180,E1 -9732.904,E2 -9732.904} C_VEL
LIN {X 0,Y 425.362,Z 463.499,A -85,B 0,C 180,E1 -9736.605,E2 -9736.605} C_VEL
LIN {X 0,Y 425.329,Z 463.505,A -85,B 0,C 180,E1 -9739.636,E2 -9739.636} C_VEL
LIN {X 0,Y 425.308,Z 463.509,A -85,B 0,C 180,E1 -9743.365,E2 -9743.365} C_VEL
LIN {X 0,Y 425.348,Z 463.503,A -85,B 0,C 180,E1 -9746.844,E2 -9746.844} C_VEL
LIN {X 0,Y 425.291,Z 463.511,A -85,B 0,C 180,E1 -9749.719,E2 -9749.719} C_VEL
LIN {X 0,Y 425.282,Z 463.512,A -85,B 0,C 180,E1 -9753.048,E2 -9753.048} C_VEL
LIN {X 0,Y 425.285,Z 463.51,A -85,B 0,C 180,E1 -9755.929,E2 -9755.929} C_VEL
LIN {X 0,Y 425.301,Z 463.509,A -85,B 0,C 180,E1 -9759.044,E2 -9759.044} C_VEL
LIN {X 0,Y 425.331,Z 463.505,A -85,B 0,C 180,E1 -9762.646,E2 -9762.646} C_VEL
LIN {X 0,Y 425.295,Z 463.515,A -85,B 0,C 180,E1 -9765.282,E2 -9765.282} C_VEL
LIN {X 0,Y 425.349,Z 463.672,A -85,B 0,C 180,E1 -9767.927,E2 -9767.927} C_VEL
LIN {X 0,Y 426.52,Z 470.316,A -85,B 0,C 180,E1 -9771.234,E2 -9771.234} C_VEL
LIN {X 0,Y 427.323,Z 475.506,A -85,B 0,C 180,E1 -9773.696,E2 -9773.696} C_VEL
LIN {X 0,Y 427.11,Z 480.639,A -85,B 0,C 180,E1 -9775.982,E2 -9775.982} C_VEL
LIN {X 0,Y 426.492,Z 488.316,A -85,B 0,C 180,E1 -9779.281,E2 -9779.281} C_VEL
LIN {X 0,Y 425.961,Z 496.005,A -85,B 0,C 180,E1 -9782.485,E2 -9782.485} C_VEL
LIN {X 0,Y 425.448,Z 503.682,A -85,B 0,C 180,E1 -9785.608,E2 -9785.608} C_VEL
LIN {X 0,Y 425.002,Z 512.637,A -85,B 0,C 180,E1 -9789.174,E2 -9789.174} C_VEL
LIN {X 0,Y 424.699,Z 521.588,A -85,B 0,C 180,E1 -9792.671,E2 -9792.671} C_VEL
LIN {X 0,Y 424.658,Z 522.982,A -85,B 0,C 180,E1 -9793.209,E2 -9793.209} C_VEL
LIN {X 0,Y 426.63,Z 536.919,A -85,B 0,C 180,E1 -9793.737,E2 -9793.737} C_VEL
LIN {X 0,Y 428.127,Z 549.86,A -85,B 0,C 180,E1 -9794.407,E2 -9794.407} C_VEL
LIN {X 0,Y 427.404,Z 562.961,A -85,B 0,C 180,E1 -9795.234,E2 -9795.234} C_VEL
LIN {X 0,Y 426.755,Z 574.268,A -85,B 0,C 180,E1 -9796.163,E2 -9796.163} C_VEL
LIN {X 0,Y 426.112,Z 584.964,A -85,B 0,C 180,E1 -9797.256,E2 -9797.256} C_VEL
LIN {X 0,Y 425.591,Z 593.583,A -85,B 0,C 180,E1 -9798.329,E2 -9798.329} C_VEL
LIN {X 0,Y 425.049,Z 601.552,A -85,B 0,C 180,E1 -9799.521,E2 -9799.521} C_VEL
LIN {X 0,Y 424.658,Z 609.37,A -85,B 0,C 180,E1 -9800.954,E2 -9800.954} C_VEL
LIN {X 0,Y 424.385,Z 615.629,A -85,B 0,C 180,E1 -9802.387,E2 -9802.387} C_VEL
LIN {X 0,Y 424.279,Z 620.099,A -85,B 0,C 180,E1 -9803.656,E2 -9803.656} C_VEL
LIN {X 0,Y 424.223,Z 624.395,A -85,B 0,C 180,E1 -9805.249,E2 -9805.249} C_VEL
LIN {X 0,Y 424.147,Z 626.338,A -85,B 0,C 180,E1 -9806.2,E2 -9806.2} C_VEL
LIN {X 0,Y 424.246,Z 627.851,A -85,B 0,C 180,E1 -9807.152,E2 -9807.152} C_VEL
LIN {X 0,Y 424.207,Z 628.884,A -85,B 0,C 180,E1 -9808.101,E2 -9808.101} C_VEL
LIN {X 0,Y 424.202,Z 629.509,A -85,B 0,C 180,E1 -9809.051,E2 -9809.051} C_VEL
LIN {X 0,Y 424.218,Z 629.731,A -85,B 0,C 180,E1 -9810,E2 -9810} C_VEL
LIN {X 0,Y 424.19,Z 629.522,A -85,B 0,C 180,E1 -9810.95,E2 -9810.95} C_VEL
LIN {X 0,Y 424.209,Z 628.869,A -85,B 0,C 180,E1 -9811.899,E2 -9811.899} C_VEL
LIN {X 0,Y 424.235,Z 627.81,A -85,B 0,C 180,E1 -9812.849,E2 -9812.849} C_VEL
LIN {X 0,Y 424.152,Z 626.331,A -85,B 0,C 180,E1 -9813.8,E2 -9813.8} C_VEL
LIN {X 0,Y 424.237,Z 623.249,A -85,B 0,C 180,E1 -9815.228,E2 -9815.228} C_VEL
LIN {X 0,Y 424.3,Z 619.089,A -85,B 0,C 180,E1 -9816.658,E2 -9816.658} C_VEL
LIN {X 0,Y 424.532,Z 612.736,A -85,B 0,C 180,E1 -9818.329,E2 -9818.329} C_VEL
LIN {X 0,Y 424.854,Z 605.826,A -85,B 0,C 180,E1 -9819.762,E2 -9819.762} C_VEL
LIN {X 0,Y 425.376,Z 597.308,A -85,B 0,C 180,E1 -9821.194,E2 -9821.194} C_VEL
LIN {X 0,Y 425.887,Z 588.658,A -85,B 0,C 180,E1 -9822.388,E2 -9822.388} C_VEL
LIN {X 0,Y 426.594,Z 578.011,A -85,B 0,C 180,E1 -9823.589,E2 -9823.589} C_VEL
LIN {X 0,Y 427.426,Z 566.464,A -85,B 0,C 180,E1 -9824.644,E2 -9824.644} C_VEL
LIN {X 0,Y 428.205,Z 555.156,A -85,B 0,C 180,E1 -9825.469,E2 -9825.469} C_VEL
LIN {X 0,Y 428.242,Z 548.37,A -85,B 0,C 180,E1 -9825.895,E2 -9825.895} C_VEL
LIN {X 0,Y 427.014,Z 534.485,A -85,B 0,C 180,E1 -9826.661,E2 -9826.661} C_VEL
LIN {X 0,Y 424.953,Z 522.164,A -85,B 0,C 180,E1 -9827.216,E2 -9827.216} C_VEL
LIN {X 0,Y 424.635,Z 519.993,A -85,B 0,C 180,E1 -9827.332,E2 -9827.332} C_VEL
LIN {X 0,Y 424.922,Z 510.95,A -85,B 0,C 180,E1 -9830.83,E2 -9830.83} C_VEL
LIN {X 0,Y 425.305,Z 502.159,A -85,B 0,C 180,E1 -9834.401,E2 -9834.401} C_VEL
LIN {X 0,Y 425.827,Z 494.923,A -85,B 0,C 180,E1 -9837.524,E2 -9837.524} C_VEL
LIN {X 0,Y 426.492,Z 487.496,A -85,B 0,C 180,E1 -9841.031,E2 -9841.031} C_VEL
LIN {X 0,Y 427.197,Z 481.859,A -85,B 0,C 180,E1 -9844.011,E2 -9844.011} C_VEL
LIN {X 0,Y 427.529,Z 478.039,A -85,B 0,C 180,E1 -9846.342,E2 -9846.342} C_VEL
LIN {X 0,Y 427.306,Z 474.87,A -85,B 0,C 180,E1 -9848.682,E2 -9848.682} C_VEL
LIN {X 0,Y 426.82,Z 472.197,A -85,B 0,C 180,E1 -9851.196,E2 -9851.196} C_VEL
LIN {X 0,Y 426.465,Z 470.148,A -85,B 0,C 180,E1 -9853.801,E2 -9853.801} C_VEL
LIN {X 0,Y 426.244,Z 468.783,A -85,B 0,C 180,E1 -9856.509,E2 -9856.509} C_VEL
LIN {X 0,Y 426.057,Z 468.151,A -85,B 0,C 180,E1 -9859.358,E2 -9859.358} C_VEL
LIN {X 0,Y 426.038,Z 468.222,A -85,B 0,C 180,E1 -9862.385,E2 -9862.385} C_VEL
LIN {X 0,Y 425.95,Z 468.743,A -85,B 0,C 180,E1 -9864.726,E2 -9864.726} C_VEL
LIN {X 0,Y 425.682,Z 470.062,A -85,B 0,C 180,E1 -9868.108,E2 -9868.108} C_VEL
LIN {X 0,Y 425.393,Z 471.802,A -85,B 0,C 180,E1 -9871.372,E2 -9871.372} C_VEL
LIN {X 0,Y 425.105,Z 473.831,A -85,B 0,C 180,E1 -9874.543,E2 -9874.543} C_VEL
LIN {X 0,Y 424.92,Z 476.201,A -85,B 0,C 180,E1 -9877.853,E2 -9877.853} C_VEL
LIN {X 0,Y 424.83,Z 478.404,A -85,B 0,C 180,E1 -9880.679,E2 -9880.679} C_VEL
LIN {X 0,Y 424.738,Z 480.197,A -85,B 0,C 180,E1 -9882.841,E2 -9882.841} C_VEL
LIN {X 0,Y 428.594,Z 493.149,A -85,B 0,C 180,E1 -9883.593,E2 -9883.593} C_VEL
LIN {X 0,Y 429.633,Z 498.307,A -85,B 0,C 180,E1 -9883.915,E2 -9883.915} C_VEL
LIN {X 0,Y 429.027,Z 511.04,A -85,B 0,C 180,E1 -9884.684,E2 -9884.684} C_VEL
LIN {X 0,Y 428.246,Z 522.863,A -85,B 0,C 180,E1 -9885.604,E2 -9885.604} C_VEL
LIN {X 0,Y 427.494,Z 534.006,A -85,B 0,C 180,E1 -9886.694,E2 -9886.694} C_VEL
LIN {X 0,Y 426.758,Z 543.75,A -85,B 0,C 180,E1 -9887.879,E2 -9887.879} C_VEL
LIN {X 0,Y 426.044,Z 553.209,A -85,B 0,C 180,E1 -9889.305,E2 -9889.305} C_VEL
LIN {X 0,Y 425.533,Z 560.801,A -85,B 0,C 180,E1 -9890.734,E2 -9890.734} C_VEL
LIN {X 0,Y 424.993,Z 567.772,A -85,B 0,C 180,E1 -9892.398,E2 -9892.398} C_VEL
LIN {X 0,Y 424.709,Z 572.416,A -85,B 0,C 180,E1 -9893.825,E2 -9893.825} C_VEL
LIN {X 0,Y 424.568,Z 575.939,A -85,B 0,C 180,E1 -9895.253,E2 -9895.253} C_VEL
LIN {X 0,Y 424.465,Z 577.741,A -85,B 0,C 180,E1 -9896.203,E2 -9896.203} C_VEL
LIN {X 0,Y 424.357,Z 579.072,A -85,B 0,C 180,E1 -9897.152,E2 -9897.152} C_VEL
LIN {X 0,Y 424.339,Z 579.994,A -85,B 0,C 180,E1 -9898.102,E2 -9898.102} C_VEL
LIN {X 0,Y 424.254,Z 580.529,A -85,B 0,C 180,E1 -9899.051,E2 -9899.051} C_VEL
LIN {X 0,Y 424.22,Z 580.65,A -85,B 0,C 180,E1 -9900,E2 -9900} C_VEL
LIN {X 0,Y 424.255,Z 579.626,A -85,B 0,C 180,E1 -9901.899,E2 -9901.899} C_VEL
LIN {X 0,Y 424.335,Z 578.52,A -85,B 0,C 180,E1 -9902.848,E2 -9902.848} C_VEL
LIN {X 0,Y 424.399,Z 576.973,A -85,B 0,C 180,E1 -9903.798,E2 -9903.798} C_VEL
LIN {X 0,Y 424.427,Z 573.839,A -85,B 0,C 180,E1 -9905.226,E2 -9905.226} C_VEL
LIN {X 0,Y 424.772,Z 568.71,A -85,B 0,C 180,E1 -9906.914,E2 -9906.914} C_VEL
LIN {X 0,Y 425.054,Z 562.148,A -85,B 0,C 180,E1 -9908.558,E2 -9908.558} C_VEL
LIN {X 0,Y 425.471,Z 554.853,A -85,B 0,C 180,E1 -9909.988,E2 -9909.988} C_VEL
LIN {X 0,Y 426.029,Z 545.815,A -85,B 0,C 180,E1 -9911.418,E2 -9911.418} C_VEL
LIN {X 0,Y 426.64,Z 536.552,A -85,B 0,C 180,E1 -9912.608,E2 -9912.608} C_VEL
LIN {X 0,Y 427.299,Z 526.04,A -85,B 0,C 180,E1 -9913.701,E2 -9913.701} C_VEL
LIN {X 0,Y 427.83,Z 515.058,A -85,B 0,C 180,E1 -9914.63,E2 -9914.63} C_VEL
LIN {X 0,Y 428.463,Z 502.827,A -85,B 0,C 180,E1 -9915.443,E2 -9915.443} C_VEL
LIN {X 0,Y 428.486,Z 495.488,A -85,B 0,C 180,E1 -9915.84,E2 -9915.84} C_VEL
LIN {X 0,Y 425.651,Z 482.653,A -85,B 0,C 180,E1 -9916.48,E2 -9916.48} C_VEL
LIN {X 0,Y 424.349,Z 476.844,A -85,B 0,C 180,E1 -9916.724,E2 -9916.724} C_VEL
LIN {X 0,Y 424.371,Z 474.035,A -85,B 0,C 180,E1 -9919.343,E2 -9919.343} C_VEL
LIN {X 0,Y 424.386,Z 470.839,A -85,B 0,C 180,E1 -9922.389,E2 -9922.389} C_VEL
LIN {X 0,Y 424.494,Z 467.62,A -85,B 0,C 180,E1 -9925.497,E2 -9925.497} C_VEL
LIN {X 0,Y 424.559,Z 464.385,A -85,B 0,C 180,E1 -9928.69,E2 -9928.69} C_VEL
LIN {X 0,Y 424.589,Z 463.6,A -85,B 0,C 180,E1 -9929.774,E2 -9929.774} C_VEL
LIN {X 0,Y 424.949,Z 463.552,A -85,B 0,C 180,E1 -9933.078,E2 -9933.078} C_VEL
LIN {X 0,Y 425.212,Z 463.52,A -85,B 0,C 180,E1 -9935.915,E2 -9935.915} C_VEL
LIN {X 0,Y 425.297,Z 463.506,A -85,B 0,C 180,E1 -9939.043,E2 -9939.043} C_VEL
LIN {X 0,Y 425.279,Z 463.513,A -85,B 0,C 180,E1 -9942.653,E2 -9942.653} C_VEL
LIN {X 0,Y 425.266,Z 463.514,A -85,B 0,C 180,E1 -9946.044,E2 -9946.044} C_VEL
LIN {X 0,Y 425.279,Z 463.511,A -85,B 0,C 180,E1 -9948.622,E2 -9948.622} C_VEL
LIN {X 0,Y 425.318,Z 463.505,A -85,B 0,C 180,E1 -9951.103,E2 -9951.103} C_VEL
LIN {X 0,Y 425.304,Z 463.507,A -85,B 0,C 180,E1 -9954.664,E2 -9954.664} C_VEL
LIN {X 0,Y 425.27,Z 463.513,A -85,B 0,C 180,E1 -9958.073,E2 -9958.073} C_VEL
LIN {X 0,Y 425.336,Z 463.502,A -85,B 0,C 180,E1 -9961.368,E2 -9961.368} C_VEL
LIN {X 0,Y 425.301,Z 463.51,A -85,B 0,C 180,E1 -9964.555,E2 -9964.555} C_VEL
LIN {X 0,Y 425.293,Z 463.508,A -85,B 0,C 180,E1 -9967.661,E2 -9967.661} C_VEL
LIN {X 0,Y 425.368,Z 463.5,A -85,B 0,C 180,E1 -9970.704,E2 -9970.704} C_VEL
LIN {X 0,Y 425.394,Z 463.496,A -85,B 0,C 180,E1 -9973.688,E2 -9973.688} C_VEL
LIN {X 0,Y 425.418,Z 463.495,A -85,B 0,C 180,E1 -9977.598,E2 -9977.598} C_VEL
LIN {X 0,Y 425.441,Z 463.489,A -85,B 0,C 180,E1 -9981.45,E2 -9981.45} C_VEL
LIN {X 0,Y 425.557,Z 463.476,A -85,B 0,C 180,E1 -9984.313,E2 -9984.313} C_VEL
LIN {X 0,Y 425.579,Z 463.476,A -85,B 0,C 180,E1 -9988.107,E2 -9988.107} C_VEL
LIN {X 0,Y 425.707,Z 463.46,A -85,B 0,C 180,E1 -9990,E2 -9990} C_VEL
LIN {X 0,Y 425.55,Z 463.476,A -85,B 0,C 180,E1 -9992.84,E2 -9992.84} C_VEL
LIN {X 0,Y 425.431,Z 463.489,A -85,B 0,C 180,E1 -9995.145,E2 -9995.145} C_VEL
LIN {X 0,Y 424.862,Z 463.565,A -85,B 0,C 180,E1 -9995.936,E2 -9995.936} C_VEL
LIN {X 0,Y 422.013,Z 463.916,A -85,B 0,C 180,E1 -9997.22,E2 -9997.22} C_VEL
LIN {X 0,Y 419.53,Z 464.227,A -85,B 0,C 180,E1 -9998.257,E2 -9998.257} C_VEL
LIN {X 0,Y 418.446,Z 464.361,A -85,B 0,C 180,E1 -9999.059,E2 -9999.059} C_VEL
LIN {X 0,Y 418.352,Z 464.373,A -85,B 0,C 180,E1 -9999.331,E2 -9999.331} C_VEL
LIN {X 0,Y 418.351,Z 464.371,A -85,B 0,C 180,E1 -10003.001,E2 -10003.001} C_VEL
LIN {X 0,Y 418.318,Z 464.377,A -85,B 0,C 180,E1 -10006.735,E2 -10006.735} C_VEL
LIN {X 0,Y 418.276,Z 464.384,A -85,B 0,C 180,E1 -10009.79,E2 -10009.79} C_VEL
LIN {X 0,Y 418.243,Z 464.386,A -85,B 0,C 180,E1 -10012.736,E2 -10012.736} C_VEL
LIN {X 0,Y 418.275,Z 464.385,A -85,B 0,C 180,E1 -10015.904,E2 -10015.904} C_VEL
LIN {X 0,Y 418.269,Z 464.382,A -85,B 0,C 180,E1 -10019.161,E2 -10019.161} C_VEL
LIN {X 0,Y 418.261,Z 464.384,A -85,B 0,C 180,E1 -10022.844,E2 -10022.844} C_VEL
LIN {X 0,Y 418.252,Z 464.386,A -85,B 0,C 180,E1 -10026.238,E2 -10026.238} C_VEL
LIN {X 0,Y 418.255,Z 464.386,A -85,B 0,C 180,E1 -10029.681,E2 -10029.681} C_VEL
LIN {X 0,Y 418.234,Z 464.387,A -85,B 0,C 180,E1 -10032.321,E2 -10032.321} C_VEL
LIN {X 0,Y 418.242,Z 464.387,A -85,B 0,C 180,E1 -10035.109,E2 -10035.109} C_VEL
LIN {X 0,Y 418.245,Z 464.388,A -85,B 0,C 180,E1 -10037.767,E2 -10037.767} C_VEL
LIN {X 0,Y 418.254,Z 464.388,A -85,B 0,C 180,E1 -10041.558,E2 -10041.558} C_VEL
LIN {X 0,Y 418.262,Z 464.385,A -85,B 0,C 180,E1 -10045.159,E2 -10045.159} C_VEL
LIN {X 0,Y 418.247,Z 464.388,A -85,B 0,C 180,E1 -10047.472,E2 -10047.472} C_VEL
LIN {X 0,Y 418.27,Z 464.383,A -85,B 0,C 180,E1 -10050.895,E2 -10050.895} C_VEL
LIN {X 0,Y 418.272,Z 464.383,A -85,B 0,C 180,E1 -10054.096,E2 -10054.096} C_VEL
LIN {X 0,Y 418.24,Z 464.39,A -85,B 0,C 180,E1 -10057.264,E2 -10057.264} C_VEL
LIN {X 0,Y 418.285,Z 464.38,A -85,B 0,C 180,E1 -10060.364,E2 -10060.364} C_VEL
LIN {X 0,Y 418.319,Z 464.38,A -85,B 0,C 180,E1 -10063.404,E2 -10063.404} C_VEL
LIN {X 0,Y 418.347,Z 464.374,A -85,B 0,C 180,E1 -10066.999,E2 -10066.999} C_VEL
LIN {X 0,Y 418.343,Z 464.374,A -85,B 0,C 180,E1 -10070.328,E2 -10070.328} C_VEL
LIN {X 0,Y 418.495,Z 464.356,A -85,B 0,C 180,E1 -10073.249,E2 -10073.249} C_VEL
LIN {X 0,Y 418.34,Z 464.375,A -85,B 0,C 180,E1 -10075.181,E2 -10075.181} C_VEL
LIN {X 0,Y 418.546,Z 464.35,A -85,B 0,C 180,E1 -10078.075,E2 -10078.075} C_VEL
LIN {X 0,Y 418.674,Z 464.334,A -85,B 0,C 180,E1 -10080,E2 -10080} C_VEL
LIN {X 0,Y 418.502,Z 464.353,A -85,B 0,C 180,E1 -10082.888,E2 -10082.888} C_VEL
LIN {X 0,Y 418.495,Z 464.356,A -85,B 0,C 180,E1 -10086.751,E2 -10086.751} C_VEL
LIN {X 0,Y 418.341,Z 464.376,A -85,B 0,C 180,E1 -10089.671,E2 -10089.671} C_VEL
LIN {X 0,Y 418.347,Z 464.376,A -85,B 0,C 180,E1 -10093.001,E2 -10093.001} C_VEL
LIN {X 0,Y 418.313,Z 464.377,A -85,B 0,C 180,E1 -10096.736,E2 -10096.736} C_VEL
LIN {X 0,Y 418.271,Z 464.384,A -85,B 0,C 180,E1 -10099.79,E2 -10099.79} C_VEL
LIN {X 0,Y 418.238,Z 464.388,A -85,B 0,C 180,E1 -10102.736,E2 -10102.736} C_VEL
LIN {X 0,Y 418.271,Z 464.383,A -85,B 0,C 180,E1 -10105.904,E2 -10105.904} C_VEL
LIN {X 0,Y 418.265,Z 464.385,A -85,B 0,C 180,E1 -10109.162,E2 -10109.162} C_VEL
LIN {X 0,Y 418.258,Z 464.385,A -85,B 0,C 180,E1 -10112.844,E2 -10112.844} C_VEL
LIN {X 0,Y 418.249,Z 464.385,A -85,B 0,C 180,E1 -10116.239,E2 -10116.239} C_VEL
LIN {X 0,Y 418.253,Z 464.385,A -85,B 0,C 180,E1 -10119.682,E2 -10119.682} C_VEL
LIN {X 0,Y 418.284,Z 464.381,A -85,B 0,C 180,E1 -10122.329,E2 -10122.329} C_VEL
LIN {X 0,Y 418.251,Z 464.391,A -85,B 0,C 180,E1 -10125.111,E2 -10125.111} C_VEL
LIN {X 0,Y 418.311,Z 464.539,A -85,B 0,C 180,E1 -10127.667,E2 -10127.667} C_VEL
LIN {X 0,Y 419.499,Z 471.281,A -85,B 0,C 180,E1 -10131.087,E2 -10131.087} C_VEL
LIN {X 0,Y 420.265,Z 476.034,A -85,B 0,C 180,E1 -10133.388,E2 -10133.388} C_VEL
LIN {X 0,Y 420.19,Z 480.31,A -85,B 0,C 180,E1 -10135.342,E2 -10135.342} C_VEL
LIN {X 0,Y 419.558,Z 487.974,A -85,B 0,C 180,E1 -10138.716,E2 -10138.716} C_VEL
LIN {X 0,Y 418.988,Z 495.646,A -85,B 0,C 180,E1 -10141.988,E2 -10141.988} C_VEL
LIN {X 0,Y 418.443,Z 503.306,A -85,B 0,C 180,E1 -10145.173,E2 -10145.173} C_VEL
LIN {X 0,Y 418.025,Z 510.953,A -85,B 0,C 180,E1 -10148.292,E2 -10148.292} C_VEL
LIN {X 0,Y 417.708,Z 518.61,A -85,B 0,C 180,E1 -10151.357,E2 -10151.357} C_VEL
LIN {X 0,Y 417.587,Z 522.691,A -85,B 0,C 180,E1 -10152.978,E2 -10152.978} C_VEL
LIN {X 0,Y 419.593,Z 536.796,A -85,B 0,C 180,E1 -10153.518,E2 -10153.518} C_VEL
LIN {X 0,Y 421.026,Z 550.012,A -85,B 0,C 180,E1 -10154.218,E2 -10154.218} C_VEL
LIN {X 0,Y 420.53,Z 561.897,A -85,B 0,C 180,E1 -10154.987,E2 -10154.987} C_VEL
LIN {X 0,Y 419.865,Z 572.69,A -85,B 0,C 180,E1 -10155.867,E2 -10155.867} C_VEL
LIN {X 0,Y 419.246,Z 583.073,A -85,B 0,C 180,E1 -10156.92,E2 -10156.92} C_VEL
LIN {X 0,Y 418.604,Z 592.821,A -85,B 0,C 180,E1 -10158.132,E2 -10158.132} C_VEL
LIN {X 0,Y 418.012,Z 600.846,A -85,B 0,C 180,E1 -10159.342,E2 -10159.342} C_VEL
LIN {X 0,Y 417.615,Z 608.743,A -85,B 0,C 180,E1 -10160.801,E2 -10160.801} C_VEL
LIN {X 0,Y 417.332,Z 615.047,A -85,B 0,C 180,E1 -10162.258,E2 -10162.258} C_VEL
LIN {X 0,Y 417.186,Z 619.956,A -85,B 0,C 180,E1 -10163.683,E2 -10163.683} C_VEL
LIN {X 0,Y 417.156,Z 623.887,A -85,B 0,C 180,E1 -10165.168,E2 -10165.168} C_VEL
LIN {X 0,Y 417.059,Z 625.844,A -85,B 0,C 180,E1 -10166.135,E2 -10166.135} C_VEL
LIN {X 0,Y 417.156,Z 627.38,A -85,B 0,C 180,E1 -10167.103,E2 -10167.103} C_VEL
LIN {X 0,Y 417.131,Z 628.433,A -85,B 0,C 180,E1 -10168.069,E2 -10168.069} C_VEL
LIN {X 0,Y 417.118,Z 629.069,A -85,B 0,C 180,E1 -10169.035,E2 -10169.035} C_VEL
LIN {X 0,Y 417.131,Z 629.301,A -85,B 0,C 180,E1 -10170,E2 -10170} C_VEL
LIN {X 0,Y 417.107,Z 629.113,A -85,B 0,C 180,E1 -10170.966,E2 -10170.966} C_VEL
LIN {X 0,Y 417.133,Z 628.471,A -85,B 0,C 180,E1 -10171.931,E2 -10171.931} C_VEL
LIN {X 0,Y 417.147,Z 627.416,A -85,B 0,C 180,E1 -10172.897,E2 -10172.897} C_VEL
LIN {X 0,Y 417.063,Z 625.946,A -85,B 0,C 180,E1 -10173.865,E2 -10173.865} C_VEL
LIN {X 0,Y 417.149,Z 622.881,A -85,B 0,C 180,E1 -10175.317,E2 -10175.317} C_VEL
LIN {X 0,Y 417.232,Z 618.745,A -85,B 0,C 180,E1 -10176.772,E2 -10176.772} C_VEL
LIN {X 0,Y 417.488,Z 612.425,A -85,B 0,C 180,E1 -10178.471,E2 -10178.471} C_VEL
LIN {X 0,Y 417.823,Z 605.553,A -85,B 0,C 180,E1 -10179.928,E2 -10179.928} C_VEL
LIN {X 0,Y 418.389,Z 597.085,A -85,B 0,C 180,E1 -10181.384,E2 -10181.384} C_VEL
LIN {X 0,Y 418.91,Z 588.508,A -85,B 0,C 180,E1 -10182.598,E2 -10182.598} C_VEL
LIN {X 0,Y 419.731,Z 577.5,A -85,B 0,C 180,E1 -10183.866,E2 -10183.866} C_VEL
LIN {X 0,Y 420.562,Z 566.568,A -85,B 0,C 180,E1 -10184.888,E2 -10184.888} C_VEL
LIN {X 0,Y 421.394,Z 555.528,A -85,B 0,C 180,E1 -10185.725,E2 -10185.725} C_VEL
LIN {X 0,Y 421.481,Z 549.949,A -85,B 0,C 180,E1 -10186.094,E2 -10186.094} C_VEL
LIN {X 0,Y 420.298,Z 535.421,A -85,B 0,C 180,E1 -10186.943,E2 -10186.943} C_VEL
LIN {X 0,Y 418.17,Z 522.545,A -85,B 0,C 180,E1 -10187.567,E2 -10187.567} C_VEL
LIN {X 0,Y 417.577,Z 519.519,A -85,B 0,C 180,E1 -10187.698,E2 -10187.698} C_VEL
LIN {X 0,Y 417.901,Z 510.721,A -85,B 0,C 180,E1 -10191.197,E2 -10191.197} C_VEL
LIN {X 0,Y 418.32,Z 501.933,A -85,B 0,C 180,E1 -10194.875,E2 -10194.875} C_VEL
LIN {X 0,Y 418.878,Z 494.907,A -85,B 0,C 180,E1 -10198.021,E2 -10198.021} C_VEL
LIN {X 0,Y 419.694,Z 487.166,A -85,B 0,C 180,E1 -10201.835,E2 -10201.835} C_VEL
LIN {X 0,Y 420.35,Z 482.143,A -85,B 0,C 180,E1 -10204.643,E2 -10204.643} C_VEL
LIN {X 0,Y 420.55,Z 478.558,A -85,B 0,C 180,E1 -10206.986,E2 -10206.986} C_VEL
LIN {X 0,Y 420.446,Z 476.935,A -85,B 0,C 180,E1 -10208.221,E2 -10208.221} C_VEL
LIN {X 0,Y 419.906,Z 473.798,A -85,B 0,C 180,E1 -10211.134,E2 -10211.134} C_VEL
LIN {X 0,Y 419.538,Z 471.629,A -85,B 0,C 180,E1 -10213.919,E2 -10213.919} C_VEL
LIN {X 0,Y 419.322,Z 470.292,A -85,B 0,C 180,E1 -10216.593,E2 -10216.593} C_VEL
LIN {X 0,Y 419.13,Z 469.672,A -85,B 0,C 180,E1 -10219.16,E2 -10219.16} C_VEL
LIN {X 0,Y 419.047,Z 469.61,A -85,B 0,C 180,E1 -10222.023,E2 -10222.023} C_VEL
LIN {X 0,Y 419.025,Z 469.931,A -85,B 0,C 180,E1 -10224.054,E2 -10224.054} C_VEL
LIN {X 0,Y 418.78,Z 470.881,A -85,B 0,C 180,E1 -10227.046,E2 -10227.046} C_VEL
LIN {X 0,Y 418.515,Z 472.104,A -85,B 0,C 180,E1 -10229.75,E2 -10229.75} C_VEL
LIN {X 0,Y 418.221,Z 473.963,A -85,B 0,C 180,E1 -10233.017,E2 -10233.017} C_VEL
LIN {X 0,Y 418.018,Z 476.046,A -85,B 0,C 180,E1 -10236.203,E2 -10236.203} C_VEL
LIN {X 0,Y 417.802,Z 478.333,A -85,B 0,C 180,E1 -10239.314,E2 -10239.314} C_VEL
LIN {X 0,Y 417.699,Z 480.811,A -85,B 0,C 180,E1 -10242.447,E2 -10242.447} C_VEL
LIN {X 0,Y 421.698,Z 493.709,A -85,B 0,C 180,E1 -10243.24,E2 -10243.24} C_VEL
LIN {X 0,Y 422.948,Z 500.152,A -85,B 0,C 180,E1 -10243.654,E2 -10243.654} C_VEL
LIN {X 0,Y 422.311,Z 512.489,A -85,B 0,C 180,E1 -10244.434,E2 -10244.434} C_VEL
LIN {X 0,Y 421.469,Z 523.897,A -85,B 0,C 180,E1 -10245.355,E2 -10245.355} C_VEL
LIN {X 0,Y 420.649,Z 534.96,A -85,B 0,C 180,E1 -10246.473,E2 -10246.473} C_VEL
LIN {X 0,Y 419.876,Z 544.571,A -85,B 0,C 180,E1 -10247.678,E2 -10247.678} C_VEL
LIN {X 0,Y 419.11,Z 553.978,A -85,B 0,C 180,E1 -10249.126,E2 -10249.126} C_VEL
LIN {X 0,Y 418.571,Z 561.5,A -85,B 0,C 180,E1 -10250.578,E2 -10250.578} C_VEL
LIN {X 0,Y 417.98,Z 568.418,A -85,B 0,C 180,E1 -10252.27,E2 -10252.27} C_VEL
LIN {X 0,Y 417.679,Z 573,A -85,B 0,C 180,E1 -10253.721,E2 -10253.721} C_VEL
LIN {X 0,Y 417.51,Z 576.475,A -85,B 0,C 180,E1 -10255.172,E2 -10255.172} C_VEL
LIN {X 0,Y 417.416,Z 578.247,A -85,B 0,C 180,E1 -10256.139,E2 -10256.139} C_VEL
LIN {X 0,Y 417.292,Z 579.558,A -85,B 0,C 180,E1 -10257.104,E2 -10257.104} C_VEL
LIN {X 0,Y 417.256,Z 580.465,A -85,B 0,C 180,E1 -10258.07,E2 -10258.07} C_VEL
LIN {X 0,Y 417.182,Z 580.982,A -85,B 0,C 180,E1 -10259.035,E2 -10259.035} C_VEL
LIN {X 0,Y 417.133,Z 581.07,A -85,B 0,C 180,E1 -10260,E2 -10260} C_VEL
LIN {X 0,Y 417.123,Z 580.735,A -85,B 0,C 180,E1 -10260.966,E2 -10260.966} C_VEL
LIN {X 0,Y 417.179,Z 580.002,A -85,B 0,C 180,E1 -10261.931,E2 -10261.931} C_VEL
LIN {X 0,Y 417.269,Z 578.872,A -85,B 0,C 180,E1 -10262.897,E2 -10262.897} C_VEL
LIN {X 0,Y 417.302,Z 576.35,A -85,B 0,C 180,E1 -10264.347,E2 -10264.347} C_VEL
LIN {X 0,Y 417.473,Z 572.811,A -85,B 0,C 180,E1 -10265.797,E2 -10265.797} C_VEL
LIN {X 0,Y 417.716,Z 568.169,A -85,B 0,C 180,E1 -10267.249,E2 -10267.249} C_VEL
LIN {X 0,Y 418.077,Z 561.132,A -85,B 0,C 180,E1 -10268.946,E2 -10268.946} C_VEL
LIN {X 0,Y 418.55,Z 553.524,A -85,B 0,C 180,E1 -10270.4,E2 -10270.4} C_VEL
LIN {X 0,Y 419.038,Z 545.782,A -85,B 0,C 180,E1 -10271.611,E2 -10271.611} C_VEL
LIN {X 0,Y 419.798,Z 535.325,A -85,B 0,C 180,E1 -10272.939,E2 -10272.939} C_VEL
LIN {X 0,Y 420.398,Z 523.971,A -85,B 0,C 180,E1 -10274.104,E2 -10274.104} C_VEL
LIN {X 0,Y 420.98,Z 513.03,A -85,B 0,C 180,E1 -10274.997,E2 -10274.997} C_VEL
LIN {X 0,Y 421.648,Z 500.824,A -85,B 0,C 180,E1 -10275.776,E2 -10275.776} C_VEL
LIN {X 0,Y 421.449,Z 496.058,A -85,B 0,C 180,E1 -10276.041,E2 -10276.041} C_VEL
LIN {X 0,Y 418.52,Z 482.963,A -85,B 0,C 180,E1 -10276.714,E2 -10276.714} C_VEL
LIN {X 0,Y 417.265,Z 477.198,A -85,B 0,C 180,E1 -10276.953,E2 -10276.953} C_VEL
LIN {X 0,Y 417.301,Z 474.29,A -85,B 0,C 180,E1 -10279.684,E2 -10279.684} C_VEL
LIN {X 0,Y 417.318,Z 471.053,A -85,B 0,C 180,E1 -10282.789,E2 -10282.789} C_VEL
LIN {X 0,Y 417.427,Z 467.801,A -85,B 0,C 180,E1 -10285.961,E2 -10285.961} C_VEL
LIN {X 0,Y 417.5,Z 464.533,A -85,B 0,C 180,E1 -10289.221,E2 -10289.221} C_VEL
LIN {X 0,Y 417.878,Z 464.435,A -85,B 0,C 180,E1 -10292.561,E2 -10292.561} C_VEL
LIN {X 0,Y 418.118,Z 464.403,A -85,B 0,C 180,E1 -10294.855,E2 -10294.855} C_VEL
LIN {X 0,Y 418.229,Z 464.388,A -85,B 0,C 180,E1 -10297.833,E2 -10297.833} C_VEL
LIN {X 0,Y 418.226,Z 464.389,A -85,B 0,C 180,E1 -10300.948,E2 -10300.948} C_VEL
LIN {X 0,Y 418.214,Z 464.391,A -85,B 0,C 180,E1 -10303.73,E2 -10303.73} C_VEL
LIN {X 0,Y 418.214,Z 464.392,A -85,B 0,C 180,E1 -10306.449,E2 -10306.449} C_VEL
LIN {X 0,Y 418.228,Z 464.388,A -85,B 0,C 180,E1 -10309.13,E2 -10309.13} C_VEL
LIN {X 0,Y 418.238,Z 464.39,A -85,B 0,C 180,E1 -10312.166,E2 -10312.166} C_VEL
LIN {X 0,Y 418.27,Z 464.383,A -85,B 0,C 180,E1 -10315.42,E2 -10315.42} C_VEL
LIN {X 0,Y 418.217,Z 464.391,A -85,B 0,C 180,E1 -10318.604,E2 -10318.604} C_VEL
LIN {X 0,Y 418.297,Z 464.383,A -85,B 0,C 180,E1 -10321.937,E2 -10321.937} C_VEL
LIN {X 0,Y 418.295,Z 464.379,A -85,B 0,C 180,E1 -10325.163,E2 -10325.163} C_VEL
LIN {X 0,Y 418.24,Z 464.388,A -85,B 0,C 180,E1 -10328.304,E2 -10328.304} C_VEL
LIN {X 0,Y 418.289,Z 464.381,A -85,B 0,C 180,E1 -10331.383,E2 -10331.383} C_VEL
LIN {X 0,Y 418.308,Z 464.379,A -85,B 0,C 180,E1 -10334.406,E2 -10334.406} C_VEL
LIN {X 0,Y 418.361,Z 464.372,A -85,B 0,C 180,E1 -10337.386,E2 -10337.386} C_VEL
LIN {X 0,Y 418.344,Z 464.376,A -85,B 0,C 180,E1 -10340.328,E2 -10340.328} C_VEL
LIN {X 0,Y 418.48,Z 464.356,A -85,B 0,C 180,E1 -10343.249,E2 -10343.249} C_VEL
LIN {X 0,Y 418.344,Z 464.374,A -85,B 0,C 180,E1 -10345.181,E2 -10345.181} C_VEL
LIN {X 0,Y 418.548,Z 464.352,A -85,B 0,C 180,E1 -10348.075,E2 -10348.075} C_VEL
LIN {X 0,Y 418.677,Z 464.335,A -85,B 0,C 180,E1 -10350,E2 -10350} C_VEL
LIN {X 0,Y 418.506,Z 464.354,A -85,B 0,C 180,E1 -10352.888,E2 -10352.888} C_VEL
LIN {X 0,Y 418.504,Z 464.356,A -85,B 0,C 180,E1 -10355.783,E2 -10355.783} C_VEL
LIN {X 0,Y 418.402,Z 464.367,A -85,B 0,C 180,E1 -10358.695,E2 -10358.695} C_VEL
LIN {X 0,Y 418.352,Z 464.373,A -85,B 0,C 180,E1 -10359.331,E2 -10359.331} C_VEL
LIN {X 0,Y 417.675,Z 464.459,A -85,B 0,C 180,E1 -10360.135,E2 -10360.135} C_VEL
LIN {X 0,Y 414.828,Z 464.813,A -85,B 0,C 180,E1 -10361.44,E2 -10361.44} C_VEL
LIN {X 0,Y 412.415,Z 465.112,A -85,B 0,C 180,E1 -10362.494,E2 -10362.494} C_VEL
LIN {X 0,Y 411.364,Z 465.242,A -85,B 0,C 180,E1 -10363.309,E2 -10363.309} C_VEL
LIN {X 0,Y 411.27,Z 465.256,A -85,B 0,C 180,E1 -10363.585,E2 -10363.585} C_VEL
LIN {X 0,Y 411.262,Z 465.256,A -85,B 0,C 180,E1 -10366.888,E2 -10366.888} C_VEL
LIN {X 0,Y 411.235,Z 465.263,A -85,B 0,C 180,E1 -10369.986,E2 -10369.986} C_VEL
LIN {X 0,Y 411.208,Z 465.263,A -85,B 0,C 180,E1 -10373.147,E2 -10373.147} C_VEL
LIN {X 0,Y 411.242,Z 465.259,A -85,B 0,C 180,E1 -10376.38,E2 -10376.38} C_VEL
LIN {X 0,Y 411.204,Z 465.266,A -85,B 0,C 180,E1 -10379.712,E2 -10379.712} C_VEL
LIN {X 0,Y 411.21,Z 465.263,A -85,B 0,C 180,E1 -10383.155,E2 -10383.155} C_VEL
LIN {X 0,Y 411.199,Z 465.263,A -85,B 0,C 180,E1 -10386.553,E2 -10386.553} C_VEL
LIN {X 0,Y 411.219,Z 465.263,A -85,B 0,C 180,E1 -10389.728,E2 -10389.728} C_VEL
LIN {X 0,Y 411.178,Z 465.265,A -85,B 0,C 180,E1 -10393.133,E2 -10393.133} C_VEL
LIN {X 0,Y 411.175,Z 465.268,A -85,B 0,C 180,E1 -10395.88,E2 -10395.88} C_VEL
LIN {X 0,Y 411.166,Z 465.266,A -85,B 0,C 180,E1 -10398.771,E2 -10398.771} C_VEL
LIN {X 0,Y 411.199,Z 465.265,A -85,B 0,C 180,E1 -10402.026,E2 -10402.026} C_VEL
LIN {X 0,Y 411.209,Z 465.265,A -85,B 0,C 180,E1 -10405.666,E2 -10405.666} C_VEL
